LIN {X 0,Y 284.664,Z 673.734,A -85,B 0,C 180,E1 -17037.975,E2 -17037.975} C_VEL
LIN {X 0,Y 285.259,Z 669.776,A -85,B 0,C 180,E1 -17041.157,E2 -17041.157} C_VEL
LIN {X 0,Y 285.946,Z 665.881,A -85,B 0,C 180,E1 -17044.423,E2 -17044.423} C_VEL
LIN {X 0,Y 286.19,Z 663.974,A -85,B 0,C 180,E1 -17046.113,E2 -17046.113} C_VEL
LIN {X 0,Y 286.242,Z 661.735,A -85,B 0,C 180,E1 -17048.216,E2 -17048.216} C_VEL
LIN {X 0,Y 285.887,Z 658.472,A -85,B 0,C 180,E1 -17051.587,E2 -17051.587} C_VEL
LIN {X 0,Y 285.336,Z 655.024,A -85,B 0,C 180,E1 -17055.585,E2 -17055.585} C_VEL
LIN {X 0,Y 284.965,Z 653.006,A -85,B 0,C 180,E1 -17058.249,E2 -17058.249} C_VEL
LIN {X 0,Y 284.54,Z 650.367,A -85,B 0,C 180,E1 -17062.222,E2 -17062.222} C_VEL
LIN {X 0,Y 284.343,Z 649.066,A -85,B 0,C 180,E1 -17064.652,E2 -17064.652} C_VEL
LIN {X 0,Y 284.295,Z 649.074,A -85,B 0,C 180,E1 -17068.726,E2 -17068.726} C_VEL
LIN {X 0,Y 284.396,Z 649.061,A -85,B 0,C 180,E1 -17072.828,E2 -17072.828} C_VEL
LIN {X 0,Y 284.368,Z 649.062,A -85,B 0,C 180,E1 -17076.707,E2 -17076.707} C_VEL
LIN {X 0,Y 284.406,Z 649.059,A -85,B 0,C 180,E1 -17081.262,E2 -17081.262} C_VEL
LIN {X 0,Y 284.494,Z 649.049,A -85,B 0,C 180,E1 -17084.459,E2 -17084.459} C_VEL
LIN {X 0,Y 284.491,Z 649.049,A -85,B 0,C 180,E1 -17088.602,E2 -17088.602} C_VEL
LIN {X 0,Y 284.661,Z 649.027,A -85,B 0,C 180,E1 -17091.481,E2 -17091.481} C_VEL
LIN {X 0,Y 284.604,Z 649.032,A -85,B 0,C 180,E1 -17094.331,E2 -17094.331} C_VEL
LIN {X 0,Y 284.858,Z 649.081,A -85,B 0,C 180,E1 -17098.586,E2 -17098.586} C_VEL
LIN {X 0,Y 285.092,Z 650.526,A -85,B 0,C 180,E1 -17101.413,E2 -17101.413} C_VEL
LIN {X 0,Y 285.18,Z 653.062,A -85,B 0,C 180,E1 -17105.657,E2 -17105.657} C_VEL
LIN {X 0,Y 285.314,Z 654.934,A -85,B 0,C 180,E1 -17108.499,E2 -17108.499} C_VEL
LIN {X 0,Y 284.959,Z 657.078,A -85,B 0,C 180,E1 -17111.38,E2 -17111.38} C_VEL
LIN {X 0,Y 284.349,Z 660.574,A -85,B 0,C 180,E1 -17115.776,E2 -17115.776} C_VEL
LIN {X 0,Y 284.199,Z 661.864,A -85,B 0,C 180,E1 -17117.124,E2 -17117.124} C_VEL
LIN {X 0,Y 285.245,Z 664.861,A -85,B 0,C 180,E1 -17117.428,E2 -17117.428} C_VEL
LIN {X 0,Y 288.856,Z 674.081,A -85,B 0,C 180,E1 -17118.485,E2 -17118.485} C_VEL
LIN {X 0,Y 292.289,Z 685.508,A -85,B 0,C 180,E1 -17119.855,E2 -17119.855} C_VEL
LIN {X 0,Y 294.405,Z 695.768,A -85,B 0,C 180,E1 -17121.173,E2 -17121.173} C_VEL
LIN {X 0,Y 295.274,Z 703.306,A -85,B 0,C 180,E1 -17122.192,E2 -17122.192} C_VEL
LIN {X 0,Y 293.386,Z 714.511,A -85,B 0,C 180,E1 -17123.656,E2 -17123.656} C_VEL
LIN {X 0,Y 291.318,Z 724.902,A -85,B 0,C 180,E1 -17125.354,E2 -17125.354} C_VEL
LIN {X 0,Y 289.305,Z 733.961,A -85,B 0,C 180,E1 -17127.193,E2 -17127.193} C_VEL
LIN {X 0,Y 287.446,Z 742.096,A -85,B 0,C 180,E1 -17129.275,E2 -17129.275} C_VEL
LIN {X 0,Y 285.831,Z 749.014,A -85,B 0,C 180,E1 -17131.5,E2 -17131.5} C_VEL
LIN {X 0,Y 284.513,Z 754.577,A -85,B 0,C 180,E1 -17133.778,E2 -17133.778} C_VEL
LIN {X 0,Y 283.654,Z 758.382,A -85,B 0,C 180,E1 -17135.814,E2 -17135.814} C_VEL
LIN {X 0,Y 282.915,Z 761.858,A -85,B 0,C 180,E1 -17138.392,E2 -17138.392} C_VEL
LIN {X 0,Y 282.479,Z 763.537,A -85,B 0,C 180,E1 -17140.306,E2 -17140.306} C_VEL
LIN {X 0,Y 282.248,Z 764.48,A -85,B 0,C 180,E1 -17142.245,E2 -17142.245} C_VEL
LIN {X 0,Y 282.092,Z 764.707,A -85,B 0,C 180,E1 -17144.234,E2 -17144.234} C_VEL
LIN {X 0,Y 282.099,Z 764.15,A -85,B 0,C 180,E1 -17146.26,E2 -17146.26} C_VEL
LIN {X 0,Y 282.277,Z 762.717,A -85,B 0,C 180,E1 -17148.325,E2 -17148.325} C_VEL
LIN {X 0,Y 282.558,Z 760.336,A -85,B 0,C 180,E1 -17150.449,E2 -17150.449} C_VEL
LIN {X 0,Y 282.955,Z 756.862,A -85,B 0,C 180,E1 -17152.638,E2 -17152.638} C_VEL
LIN {X 0,Y 283.587,Z 752.143,A -85,B 0,C 180,E1 -17154.868,E2 -17154.868} C_VEL
LIN {X 0,Y 284.477,Z 745.924,A -85,B 0,C 180,E1 -17157.137,E2 -17157.137} C_VEL
LIN {X 0,Y 285.721,Z 737.947,A -85,B 0,C 180,E1 -17159.419,E2 -17159.419} C_VEL
LIN {X 0,Y 286.896,Z 730.138,A -85,B 0,C 180,E1 -17161.224,E2 -17161.224} C_VEL
LIN {X 0,Y 288.359,Z 720.685,A -85,B 0,C 180,E1 -17163.004,E2 -17163.004} C_VEL
LIN {X 0,Y 289.993,Z 709.239,A -85,B 0,C 180,E1 -17164.713,E2 -17164.713} C_VEL
LIN {X 0,Y 291.243,Z 698.743,A -85,B 0,C 180,E1 -17165.97,E2 -17165.97} C_VEL
LIN {X 0,Y 289.669,Z 688.156,A -85,B 0,C 180,E1 -17167.157,E2 -17167.157} C_VEL
LIN {X 0,Y 287.141,Z 675.561,A -85,B 0,C 180,E1 -17168.319,E2 -17168.319} C_VEL
LIN {X 0,Y 283.658,Z 661.926,A -85,B 0,C 180,E1 -17169.325,E2 -17169.325} C_VEL
LIN {X 0,Y 283.257,Z 660.019,A -85,B 0,C 180,E1 -17169.437,E2 -17169.437} C_VEL
LIN {X 0,Y 283.549,Z 656.758,A -85,B 0,C 180,E1 -17172.696,E2 -17172.696} C_VEL
LIN {X 0,Y 283.905,Z 653.867,A -85,B 0,C 180,E1 -17175.667,E2 -17175.667} C_VEL
LIN {X 0,Y 284.361,Z 649.706,A -85,B 0,C 180,E1 -17180.037,E2 -17180.037} C_VEL
LIN {X 0,Y 284.468,Z 649.053,A -85,B 0,C 180,E1 -17180.81,E2 -17180.81} C_VEL
LIN {X 0,Y 284.669,Z 649.026,A -85,B 0,C 180,E1 -17182.909,E2 -17182.909} C_VEL
LIN {X 0,Y 284.859,Z 649.001,A -85,B 0,C 180,E1 -17188.586,E2 -17188.586} C_VEL
LIN {X 0,Y 284.859,Z 648.998,A -85,B 0,C 180,E1 -17191.413,E2 -17191.413} C_VEL
LIN {X 0,Y 284.575,Z 649.035,A -85,B 0,C 180,E1 -17195.669,E2 -17195.669} C_VEL
LIN {X 0,Y 284.438,Z 649.054,A -85,B 0,C 180,E1 -17198.758,E2 -17198.758} C_VEL
LIN {X 0,Y 283.86,Z 649.144,A -85,B 0,C 180,E1 -17202.148,E2 -17202.148} C_VEL
LIN {X 0,Y 283.426,Z 653.771,A -85,B 0,C 180,E1 -17205.828,E2 -17205.828} C_VEL
LIN {X 0,Y 283.169,Z 658.716,A -85,B 0,C 180,E1 -17209.686,E2 -17209.686} C_VEL
LIN {X 0,Y 286.493,Z 672.258,A -85,B 0,C 180,E1 -17210.601,E2 -17210.601} C_VEL
LIN {X 0,Y 288.907,Z 683.729,A -85,B 0,C 180,E1 -17211.587,E2 -17211.587} C_VEL
LIN {X 0,Y 290.897,Z 696.161,A -85,B 0,C 180,E1 -17212.904,E2 -17212.904} C_VEL
LIN {X 0,Y 290.964,Z 700.386,A -85,B 0,C 180,E1 -17213.384,E2 -17213.384} C_VEL
LIN {X 0,Y 289.541,Z 711.369,A -85,B 0,C 180,E1 -17214.752,E2 -17214.752} C_VEL
LIN {X 0,Y 287.993,Z 722.2,A -85,B 0,C 180,E1 -17216.446,E2 -17216.446} C_VEL
LIN {X 0,Y 286.526,Z 731.837,A -85,B 0,C 180,E1 -17218.342,E2 -17218.342} C_VEL
LIN {X 0,Y 285.193,Z 740.281,A -85,B 0,C 180,E1 -17220.401,E2 -17220.401} C_VEL
LIN {X 0,Y 284.106,Z 747.82,A -85,B 0,C 180,E1 -17222.747,E2 -17222.747} C_VEL
LIN {X 0,Y 283.266,Z 753.591,A -85,B 0,C 180,E1 -17225.04,E2 -17225.04} C_VEL
LIN {X 0,Y 282.695,Z 757.923,A -85,B 0,C 180,E1 -17227.293,E2 -17227.293} C_VEL
LIN {X 0,Y 282.283,Z 760.988,A -85,B 0,C 180,E1 -17229.483,E2 -17229.483} C_VEL
LIN {X 0,Y 282.008,Z 763.403,A -85,B 0,C 180,E1 -17232.288,E2 -17232.288} C_VEL
LIN {X 0,Y 282.031,Z 764.176,A -85,B 0,C 180,E1 -17234.245,E2 -17234.245} C_VEL
LIN {X 0,Y 282.115,Z 764.191,A -85,B 0,C 180,E1 -17236.255,E2 -17236.255} C_VEL
LIN {X 0,Y 282.358,Z 763.358,A -85,B 0,C 180,E1 -17238.305,E2 -17238.305} C_VEL
LIN {X 0,Y 282.718,Z 761.642,A -85,B 0,C 180,E1 -17240.408,E2 -17240.408} C_VEL
LIN {X 0,Y 283.379,Z 758.988,A -85,B 0,C 180,E1 -17242.524,E2 -17242.524} C_VEL
LIN {X 0,Y 284.183,Z 755.235,A -85,B 0,C 180,E1 -17244.696,E2 -17244.696} C_VEL
LIN {X 0,Y 285.511,Z 749.4,A -85,B 0,C 180,E1 -17247.211,E2 -17247.211} C_VEL
LIN {X 0,Y 287.087,Z 742.446,A -85,B 0,C 180,E1 -17249.499,E2 -17249.499} C_VEL
LIN {X 0,Y 288.904,Z 734.557,A -85,B 0,C 180,E1 -17251.563,E2 -17251.563} C_VEL
LIN {X 0,Y 290.969,Z 725.043,A -85,B 0,C 180,E1 -17253.531,E2 -17253.531} C_VEL
LIN {X 0,Y 292.926,Z 715.188,A -85,B 0,C 180,E1 -17255.167,E2 -17255.167} C_VEL
LIN {X 0,Y 294.891,Z 703.914,A -85,B 0,C 180,E1 -17256.658,E2 -17256.658} C_VEL
LIN {X 0,Y 294.933,Z 701.005,A -85,B 0,C 180,E1 -17257.033,E2 -17257.033} C_VEL
LIN {X 0,Y 293.39,Z 689.863,A -85,B 0,C 180,E1 -17258.473,E2 -17258.473} C_VEL
LIN {X 0,Y 290.907,Z 679.391,A -85,B 0,C 180,E1 -17259.725,E2 -17259.725} C_VEL
LIN {X 0,Y 286.951,Z 667.38,A -85,B 0,C 180,E1 -17261.054,E2 -17261.054} C_VEL
LIN {X 0,Y 284.148,Z 660.229,A -85,B 0,C 180,E1 -17261.804,E2 -17261.804} C_VEL
LIN {X 0,Y 284.051,Z 659.674,A -85,B 0,C 180,E1 -17261.891,E2 -17261.891} C_VEL
LIN {X 0,Y 284.171,Z 658.068,A -85,B 0,C 180,E1 -17263.229,E2 -17263.229} C_VEL
LIN {X 0,Y 283.618,Z 656.803,A -85,B 0,C 180,E1 -17264.387,E2 -17264.387} C_VEL
LIN {X 0,Y 280.968,Z 655.129,A -85,B 0,C 180,E1 -17266.295,E2 -17266.295} C_VEL
LIN {X 0,Y 278.693,Z 653.829,A -85,B 0,C 180,E1 -17267.848,E2 -17267.848} C_VEL
LIN {X 0,Y 277.735,Z 652.691,A -85,B 0,C 180,E1 -17269.04,E2 -17269.04} C_VEL
LIN {X 0,Y 277.669,Z 652.253,A -85,B 0,C 180,E1 -17269.441,E2 -17269.441} C_VEL
LIN {X 0,Y 277.548,Z 649.917,A -85,B 0,C 180,E1 -17271.628,E2 -17271.628} C_VEL
LIN {X 0,Y 277.563,Z 649.914,A -85,B 0,C 180,E1 -17274.187,E2 -17274.187} C_VEL
LIN {X 0,Y 277.82,Z 649.879,A -85,B 0,C 180,E1 -17278.55,E2 -17278.55} C_VEL
LIN {X 0,Y 277.82,Z 649.88,A -85,B 0,C 180,E1 -17281.45,E2 -17281.45} C_VEL
LIN {X 0,Y 277.65,Z 649.899,A -85,B 0,C 180,E1 -17287.271,E2 -17287.271} C_VEL
LIN {X 0,Y 277.503,Z 649.918,A -85,B 0,C 180,E1 -17290.211,E2 -17290.211} C_VEL
LIN {X 0,Y 277.431,Z 649.926,A -85,B 0,C 180,E1 -17294.674,E2 -17294.674} C_VEL
LIN {X 0,Y 277.341,Z 649.936,A -85,B 0,C 180,E1 -17299.234,E2 -17299.234} C_VEL
LIN {X 0,Y 277.316,Z 649.94,A -85,B 0,C 180,E1 -17304.171,E2 -17304.171} C_VEL
LIN {X 0,Y 277.323,Z 649.942,A -85,B 0,C 180,E1 -17307.506,E2 -17307.506} C_VEL
LIN {X 0,Y 277.269,Z 649.947,A -85,B 0,C 180,E1 -17310.482,E2 -17310.482} C_VEL
LIN {X 0,Y 277.244,Z 649.95,A -85,B 0,C 180,E1 -17313.896,E2 -17313.896} C_VEL
LIN {X 0,Y 277.265,Z 649.946,A -85,B 0,C 180,E1 -17317.47,E2 -17317.47} C_VEL
LIN {X 0,Y 277.207,Z 649.956,A -85,B 0,C 180,E1 -17321.237,E2 -17321.237} C_VEL
LIN {X 0,Y 277.273,Z 650.135,A -85,B 0,C 180,E1 -17324.659,E2 -17324.659} C_VEL
LIN {X 0,Y 278.128,Z 654.82,A -85,B 0,C 180,E1 -17328.93,E2 -17328.93} C_VEL
LIN {X 0,Y 278.627,Z 657.699,A -85,B 0,C 180,E1 -17331.438,E2 -17331.438} C_VEL
LIN {X 0,Y 278.8,Z 660.491,A -85,B 0,C 180,E1 -17333.771,E2 -17333.771} C_VEL
LIN {X 0,Y 278.36,Z 663.849,A -85,B 0,C 180,E1 -17336.427,E2 -17336.427} C_VEL
LIN {X 0,Y 277.598,Z 669.016,A -85,B 0,C 180,E1 -17340.418,E2 -17340.418} C_VEL
LIN {X 0,Y 277.426,Z 670.534,A -85,B 0,C 180,E1 -17341.447,E2 -17341.447} C_VEL
LIN {X 0,Y 278.249,Z 673.76,A -85,B 0,C 180,E1 -17341.713,E2 -17341.713} C_VEL
LIN {X 0,Y 281.779,Z 685.347,A -85,B 0,C 180,E1 -17342.86,E2 -17342.86} C_VEL
LIN {X 0,Y 284.486,Z 697.852,A -85,B 0,C 180,E1 -17344.193,E2 -17344.193} C_VEL
LIN {X 0,Y 285.824,Z 708.755,A -85,B 0,C 180,E1 -17345.475,E2 -17345.475} C_VEL
LIN {X 0,Y 286.188,Z 719.399,A -85,B 0,C 180,E1 -17346.865,E2 -17346.865} C_VEL
LIN {X 0,Y 285.951,Z 725.836,A -85,B 0,C 180,E1 -17347.798,E2 -17347.798} C_VEL
LIN {X 0,Y 283.945,Z 735.872,A -85,B 0,C 180,E1 -17349.348,E2 -17349.348} C_VEL
LIN {X 0,Y 281.936,Z 744.978,A -85,B 0,C 180,E1 -17351.092,E2 -17351.092} C_VEL
LIN {X 0,Y 280.014,Z 753.864,A -85,B 0,C 180,E1 -17353.224,E2 -17353.224} C_VEL
LIN {X 0,Y 278.44,Z 761.082,A -85,B 0,C 180,E1 -17355.381,E2 -17355.381} C_VEL
LIN {X 0,Y 277.093,Z 766.88,A -85,B 0,C 180,E1 -17357.551,E2 -17357.551} C_VEL
LIN {X 0,Y 276.211,Z 771.449,A -85,B 0,C 180,E1 -17359.741,E2 -17359.741} C_VEL
LIN {X 0,Y 275.813,Z 773.863,A -85,B 0,C 180,E1 -17361.206,E2 -17361.206} C_VEL
LIN {X 0,Y 275.509,Z 775.851,A -85,B 0,C 180,E1 -17362.673,E2 -17362.673} C_VEL
LIN {X 0,Y 275.326,Z 777.779,A -85,B 0,C 180,E1 -17364.575,E2 -17364.575} C_VEL
LIN {X 0,Y 275.265,Z 780.485,A -85,B 0,C 180,E1 -17368.538,E2 -17368.538} C_VEL
LIN {X 0,Y 275.28,Z 781.022,A -85,B 0,C 180,E1 -17370.001,E2 -17370.001} C_VEL
LIN {X 0,Y 275.262,Z 781.121,A -85,B 0,C 180,E1 -17371.464,E2 -17371.464} C_VEL
LIN {X 0,Y 275.257,Z 780.809,A -85,B 0,C 180,E1 -17372.928,E2 -17372.928} C_VEL
LIN {X 0,Y 275.379,Z 779.015,A -85,B 0,C 180,E1 -17375.86,E2 -17375.86} C_VEL
LIN {X 0,Y 275.531,Z 777.483,A -85,B 0,C 180,E1 -17377.328,E2 -17377.328} C_VEL
LIN {X 0,Y 276.016,Z 774.394,A -85,B 0,C 180,E1 -17379.527,E2 -17379.527} C_VEL
LIN {X 0,Y 276.843,Z 770.267,A -85,B 0,C 180,E1 -17381.718,E2 -17381.718} C_VEL
LIN {X 0,Y 278.211,Z 763.998,A -85,B 0,C 180,E1 -17384.259,E2 -17384.259} C_VEL
LIN {X 0,Y 279.916,Z 757.219,A -85,B 0,C 180,E1 -17386.408,E2 -17386.408} C_VEL
LIN {X 0,Y 281.667,Z 748.963,A -85,B 0,C 180,E1 -17388.53,E2 -17388.53} C_VEL
LIN {X 0,Y 283.596,Z 740.359,A -85,B 0,C 180,E1 -17390.301,E2 -17390.301} C_VEL
LIN {X 0,Y 285.822,Z 729.966,A -85,B 0,C 180,E1 -17392.023,E2 -17392.023} C_VEL
LIN {X 0,Y 286.844,Z 723.901,A -85,B 0,C 180,E1 -17392.89,E2 -17392.89} C_VEL
LIN {X 0,Y 286.621,Z 713.07,A -85,B 0,C 180,E1 -17394.404,E2 -17394.404} C_VEL
LIN {X 0,Y 285.273,Z 701.307,A -85,B 0,C 180,E1 -17395.863,E2 -17395.863} C_VEL
LIN {X 0,Y 282.516,Z 688.923,A -85,B 0,C 180,E1 -17397.285,E2 -17397.285} C_VEL
LIN {X 0,Y 279.072,Z 677.521,A -85,B 0,C 180,E1 -17398.511,E2 -17398.511} C_VEL
LIN {X 0,Y 277.896,Z 674.354,A -85,B 0,C 180,E1 -17398.849,E2 -17398.849} C_VEL
LIN {X 0,Y 277.781,Z 673.521,A -85,B 0,C 180,E1 -17398.939,E2 -17398.939} C_VEL
LIN {X 0,Y 278.409,Z 669.828,A -85,B 0,C 180,E1 -17402.014,E2 -17402.014} C_VEL
LIN {X 0,Y 279.079,Z 665.982,A -85,B 0,C 180,E1 -17405.395,E2 -17405.395} C_VEL
LIN {X 0,Y 279.227,Z 664.096,A -85,B 0,C 180,E1 -17407.162,E2 -17407.162} C_VEL
LIN {X 0,Y 279.168,Z 662.256,A -85,B 0,C 180,E1 -17409.004,E2 -17409.004} C_VEL
LIN {X 0,Y 279.005,Z 660.453,A -85,B 0,C 180,E1 -17410.915,E2 -17410.915} C_VEL
LIN {X 0,Y 278.478,Z 656.993,A -85,B 0,C 180,E1 -17414.963,E2 -17414.963} C_VEL
LIN {X 0,Y 277.945,Z 654.091,A -85,B 0,C 180,E1 -17418.896,E2 -17418.896} C_VEL
LIN {X 0,Y 277.569,Z 651.765,A -85,B 0,C 180,E1 -17422.578,E2 -17422.578} C_VEL
LIN {X 0,Y 277.249,Z 649.949,A -85,B 0,C 180,E1 -17426.104,E2 -17426.104} C_VEL
LIN {X 0,Y 277.263,Z 649.946,A -85,B 0,C 180,E1 -17429.539,E2 -17429.539} C_VEL
LIN {X 0,Y 277.358,Z 649.938,A -85,B 0,C 180,E1 -17432.864,E2 -17432.864} C_VEL
LIN {X 0,Y 277.33,Z 649.936,A -85,B 0,C 180,E1 -17436.08,E2 -17436.08} C_VEL
LIN {X 0,Y 277.347,Z 649.939,A -85,B 0,C 180,E1 -17440.766,E2 -17440.766} C_VEL
LIN {X 0,Y 277.437,Z 649.928,A -85,B 0,C 180,E1 -17445.326,E2 -17445.326} C_VEL
LIN {X 0,Y 277.509,Z 649.915,A -85,B 0,C 180,E1 -17449.789,E2 -17449.789} C_VEL
LIN {X 0,Y 277.655,Z 649.898,A -85,B 0,C 180,E1 -17452.729,E2 -17452.729} C_VEL
LIN {X 0,Y 277.701,Z 649.921,A -85,B 0,C 180,E1 -17457.099,E2 -17457.099} C_VEL
LIN {X 0,Y 278.1,Z 651.215,A -85,B 0,C 180,E1 -17460,E2 -17460} C_VEL
LIN {X 0,Y 278.154,Z 652.769,A -85,B 0,C 180,E1 -17462.897,E2 -17462.897} C_VEL
LIN {X 0,Y 278.298,Z 655.402,A -85,B 0,C 180,E1 -17467.254,E2 -17467.254} C_VEL
LIN {X 0,Y 278.127,Z 657.42,A -85,B 0,C 180,E1 -17470.188,E2 -17470.188} C_VEL
LIN {X 0,Y 277.464,Z 660.842,A -85,B 0,C 180,E1 -17474.673,E2 -17474.673} C_VEL
LIN {X 0,Y 277.293,Z 661.957,A -85,B 0,C 180,E1 -17476.092,E2 -17476.092} C_VEL
LIN {X 0,Y 278.408,Z 665.25,A -85,B 0,C 180,E1 -17476.461,E2 -17476.461} C_VEL
LIN {X 0,Y 282.09,Z 674.295,A -85,B 0,C 180,E1 -17477.583,E2 -17477.583} C_VEL
LIN {X 0,Y 285.242,Z 684.375,A -85,B 0,C 180,E1 -17478.858,E2 -17478.858} C_VEL
LIN {X 0,Y 287.762,Z 695.631,A -85,B 0,C 180,E1 -17480.367,E2 -17480.367} C_VEL
LIN {X 0,Y 288.826,Z 704.29,A -85,B 0,C 180,E1 -17481.603,E2 -17481.603} C_VEL
LIN {X 0,Y 286.967,Z 715.061,A -85,B 0,C 180,E1 -17483.07,E2 -17483.07} C_VEL
LIN {X 0,Y 284.798,Z 725.402,A -85,B 0,C 180,E1 -17484.804,E2 -17484.804} C_VEL
LIN {X 0,Y 282.782,Z 733.953,A -85,B 0,C 180,E1 -17486.574,E2 -17486.574} C_VEL
LIN {X 0,Y 280.712,Z 742.491,A -85,B 0,C 180,E1 -17488.803,E2 -17488.803} C_VEL
LIN {X 0,Y 279.007,Z 749.379,A -85,B 0,C 180,E1 -17491.081,E2 -17491.081} C_VEL
LIN {X 0,Y 277.637,Z 754.755,A -85,B 0,C 180,E1 -17493.347,E2 -17493.347} C_VEL
LIN {X 0,Y 276.601,Z 759.08,A -85,B 0,C 180,E1 -17495.76,E2 -17495.76} C_VEL
LIN {X 0,Y 275.965,Z 761.825,A -85,B 0,C 180,E1 -17497.863,E2 -17497.863} C_VEL
LIN {X 0,Y 275.429,Z 763.743,A -85,B 0,C 180,E1 -17500.048,E2 -17500.048} C_VEL
LIN {X 0,Y 275.156,Z 764.744,A -85,B 0,C 180,E1 -17502.207,E2 -17502.207} C_VEL
LIN {X 0,Y 274.99,Z 764.896,A -85,B 0,C 180,E1 -17504.307,E2 -17504.307} C_VEL
LIN {X 0,Y 275.004,Z 764.257,A -85,B 0,C 180,E1 -17506.368,E2 -17506.368} C_VEL
LIN {X 0,Y 275.184,Z 762.849,A -85,B 0,C 180,E1 -17508.392,E2 -17508.392} C_VEL
LIN {X 0,Y 275.465,Z 760.673,A -85,B 0,C 180,E1 -17510.369,E2 -17510.369} C_VEL
LIN {X 0,Y 275.781,Z 757.799,A -85,B 0,C 180,E1 -17512.293,E2 -17512.293} C_VEL
LIN {X 0,Y 276.374,Z 753.558,A -85,B 0,C 180,E1 -17514.463,E2 -17514.463} C_VEL
LIN {X 0,Y 277.188,Z 747.684,A -85,B 0,C 180,E1 -17516.794,E2 -17516.794} C_VEL
LIN {X 0,Y 278.419,Z 740.212,A -85,B 0,C 180,E1 -17519.121,E2 -17519.121} C_VEL
LIN {X 0,Y 279.643,Z 732.382,A -85,B 0,C 180,E1 -17521.067,E2 -17521.067} C_VEL
LIN {X 0,Y 281.228,Z 722.404,A -85,B 0,C 180,E1 -17523.066,E2 -17523.066} C_VEL
LIN {X 0,Y 282.664,Z 712.862,A -85,B 0,C 180,E1 -17524.611,E2 -17524.611} C_VEL
LIN {X 0,Y 284.064,Z 702.39,A -85,B 0,C 180,E1 -17525.984,E2 -17525.984} C_VEL
LIN {X 0,Y 284.159,Z 697.909,A -85,B 0,C 180,E1 -17526.515,E2 -17526.515} C_VEL
LIN {X 0,Y 282.167,Z 685.765,A -85,B 0,C 180,E1 -17527.869,E2 -17527.869} C_VEL
LIN {X 0,Y 279.45,Z 672.872,A -85,B 0,C 180,E1 -17529.047,E2 -17529.047} C_VEL
LIN {X 0,Y 276.243,Z 660.167,A -85,B 0,C 180,E1 -17529.994,E2 -17529.994} C_VEL
LIN {X 0,Y 276.595,Z 656.508,A -85,B 0,C 180,E1 -17533.769,E2 -17533.769} C_VEL
LIN {X 0,Y 276.918,Z 653.626,A -85,B 0,C 180,E1 -17536.796,E2 -17536.796} C_VEL
LIN {X 0,Y 277.495,Z 649.921,A -85,B 0,C 180,E1 -17541.02,E2 -17541.02} C_VEL
LIN {X 0,Y 277.565,Z 649.908,A -85,B 0,C 180,E1 -17544.186,E2 -17544.186} C_VEL
LIN {X 0,Y 277.825,Z 649.876,A -85,B 0,C 180,E1 -17548.55,E2 -17548.55} C_VEL
LIN {X 0,Y 277.824,Z 649.874,A -85,B 0,C 180,E1 -17551.449,E2 -17551.449} C_VEL
LIN {X 0,Y 277.54,Z 649.912,A -85,B 0,C 180,E1 -17555.813,E2 -17555.813} C_VEL
LIN {X 0,Y 277.372,Z 649.934,A -85,B 0,C 180,E1 -17558.818,E2 -17558.818} C_VEL
LIN {X 0,Y 276.837,Z 650.016,A -85,B 0,C 180,E1 -17562.089,E2 -17562.089} C_VEL
LIN {X 0,Y 276.314,Z 655.191,A -85,B 0,C 180,E1 -17566.247,E2 -17566.247} C_VEL
LIN {X 0,Y 276.146,Z 658.767,A -85,B 0,C 180,E1 -17569.127,E2 -17569.127} C_VEL
LIN {X 0,Y 279.856,Z 674,A -85,B 0,C 180,E1 -17570.235,E2 -17570.235} C_VEL
LIN {X 0,Y 282.29,Z 686.105,A -85,B 0,C 180,E1 -17571.352,E2 -17571.352} C_VEL
LIN {X 0,Y 284.209,Z 698.375,A -85,B 0,C 180,E1 -17572.729,E2 -17572.729} C_VEL
LIN {X 0,Y 283.1,Z 708.767,A -85,B 0,C 180,E1 -17573.995,E2 -17573.995} C_VEL
LIN {X 0,Y 281.417,Z 720.109,A -85,B 0,C 180,E1 -17575.723,E2 -17575.723} C_VEL
LIN {X 0,Y 280.011,Z 729.296,A -85,B 0,C 180,E1 -17577.463,E2 -17577.463} C_VEL
LIN {X 0,Y 278.625,Z 737.842,A -85,B 0,C 180,E1 -17579.462,E2 -17579.462} C_VEL
LIN {X 0,Y 277.423,Z 745.682,A -85,B 0,C 180,E1 -17581.768,E2 -17581.768} C_VEL
LIN {X 0,Y 276.548,Z 751.68,A -85,B 0,C 180,E1 -17583.992,E2 -17583.992} C_VEL
LIN {X 0,Y 275.946,Z 755.669,A -85,B 0,C 180,E1 -17585.857,E2 -17585.857} C_VEL
LIN {X 0,Y 275.32,Z 760.235,A -85,B 0,C 180,E1 -17588.711,E2 -17588.711} C_VEL
LIN {X 0,Y 274.944,Z 763.169,A -85,B 0,C 180,E1 -17591.651,E2 -17591.651} C_VEL
LIN {X 0,Y 274.933,Z 764.369,A -85,B 0,C 180,E1 -17594.295,E2 -17594.295} C_VEL
LIN {X 0,Y 275.026,Z 764.404,A -85,B 0,C 180,E1 -17596.373,E2 -17596.373} C_VEL
LIN {X 0,Y 275.275,Z 763.625,A -85,B 0,C 180,E1 -17598.409,E2 -17598.409} C_VEL
LIN {X 0,Y 275.622,Z 762.123,A -85,B 0,C 180,E1 -17600.396,E2 -17600.396} C_VEL
LIN {X 0,Y 276.256,Z 759.873,A -85,B 0,C 180,E1 -17602.369,E2 -17602.369} C_VEL
LIN {X 0,Y 276.943,Z 756.914,A -85,B 0,C 180,E1 -17604.297,E2 -17604.297} C_VEL
LIN {X 0,Y 278.024,Z 752.404,A -85,B 0,C 180,E1 -17606.53,E2 -17606.53} C_VEL
LIN {X 0,Y 279.445,Z 746.551,A -85,B 0,C 180,E1 -17608.769,E2 -17608.769} C_VEL
LIN {X 0,Y 281.274,Z 739.196,A -85,B 0,C 180,E1 -17610.987,E2 -17610.987} C_VEL
LIN {X 0,Y 283.167,Z 731.129,A -85,B 0,C 180,E1 -17612.942,E2 -17612.942} C_VEL
LIN {X 0,Y 285.089,Z 722.466,A -85,B 0,C 180,E1 -17614.638,E2 -17614.638} C_VEL
LIN {X 0,Y 287.35,Z 711.258,A -85,B 0,C 180,E1 -17616.39,E2 -17616.39} C_VEL
LIN {X 0,Y 288.529,Z 704.525,A -85,B 0,C 180,E1 -17617.27,E2 -17617.27} C_VEL
LIN {X 0,Y 287.71,Z 695.7,A -85,B 0,C 180,E1 -17618.505,E2 -17618.505} C_VEL
LIN {X 0,Y 285.726,Z 685.274,A -85,B 0,C 180,E1 -17619.857,E2 -17619.857} C_VEL
LIN {X 0,Y 282.201,Z 673.271,A -85,B 0,C 180,E1 -17621.315,E2 -17621.315} C_VEL
LIN {X 0,Y 278.28,Z 663.164,A -85,B 0,C 180,E1 -17622.501,E2 -17622.501} C_VEL
LIN {X 0,Y 277.194,Z 659.893,A -85,B 0,C 180,E1 -17622.858,E2 -17622.858} C_VEL
LIN {X 0,Y 277.622,Z 655.249,A -85,B 0,C 180,E1 -17626.83,E2 -17626.83} C_VEL
LIN {X 0,Y 277.669,Z 652.253,A -85,B 0,C 180,E1 -17629.441,E2 -17629.441} C_VEL
LIN {X 0,Y 276.986,Z 651.242,A -85,B 0,C 180,E1 -17630.631,E2 -17630.631} C_VEL
LIN {X 0,Y 275.333,Z 650.76,A -85,B 0,C 180,E1 -17631.812,E2 -17631.812} C_VEL
LIN {X 0,Y 271.5,Z 650.708,A -85,B 0,C 180,E1 -17634.203,E2 -17634.203} C_VEL
LIN {X 0,Y 270.496,Z 650.794,A -85,B 0,C 180,E1 -17635.453,E2 -17635.453} C_VEL
LIN {X 0,Y 270.452,Z 650.797,A -85,B 0,C 180,E1 -17635.876,E2 -17635.876} C_VEL
LIN {X 0,Y 270.785,Z 650.756,A -85,B 0,C 180,E1 -17638.513,E2 -17638.513} C_VEL
LIN {X 0,Y 270.785,Z 650.756,A -85,B 0,C 180,E1 -17641.487,E2 -17641.487} C_VEL
LIN {X 0,Y 270.608,Z 650.776,A -85,B 0,C 180,E1 -17647.461,E2 -17647.461} C_VEL
LIN {X 0,Y 270.438,Z 650.799,A -85,B 0,C 180,E1 -17650.481,E2 -17650.481} C_VEL
LIN {X 0,Y 270.4,Z 650.804,A -85,B 0,C 180,E1 -17655.065,E2 -17655.065} C_VEL
LIN {X 0,Y 270.298,Z 650.816,A -85,B 0,C 180,E1 -17659.756,E2 -17659.756} C_VEL
LIN {X 0,Y 270.271,Z 650.819,A -85,B 0,C 180,E1 -17664.586,E2 -17664.586} C_VEL
LIN {X 0,Y 270.267,Z 650.819,A -85,B 0,C 180,E1 -17667.909,E2 -17667.909} C_VEL
LIN {X 0,Y 270.181,Z 650.829,A -85,B 0,C 180,E1 -17671.349,E2 -17671.349} C_VEL
LIN {X 0,Y 270.199,Z 650.828,A -85,B 0,C 180,E1 -17674.906,E2 -17674.906} C_VEL
LIN {X 0,Y 270.195,Z 650.83,A -85,B 0,C 180,E1 -17678.711,E2 -17678.711} C_VEL
LIN {X 0,Y 270.169,Z 650.833,A -85,B 0,C 180,E1 -17683.251,E2 -17683.251} C_VEL
LIN {X 0,Y 270.201,Z 650.842,A -85,B 0,C 180,E1 -17684.235,E2 -17684.235} C_VEL
LIN {X 0,Y 270.815,Z 654.374,A -85,B 0,C 180,E1 -17687.568,E2 -17687.568} C_VEL
LIN {X 0,Y 271.542,Z 658.087,A -85,B 0,C 180,E1 -17690.937,E2 -17690.937} C_VEL
LIN {X 0,Y 271.755,Z 661.07,A -85,B 0,C 180,E1 -17693.502,E2 -17693.502} C_VEL
LIN {X 0,Y 271.398,Z 664.087,A -85,B 0,C 180,E1 -17695.961,E2 -17695.961} C_VEL
LIN {X 0,Y 270.547,Z 669.692,A -85,B 0,C 180,E1 -17700.366,E2 -17700.366} C_VEL
LIN {X 0,Y 271.416,Z 673.063,A -85,B 0,C 180,E1 -17700.657,E2 -17700.657} C_VEL
LIN {X 0,Y 274.431,Z 682.408,A -85,B 0,C 180,E1 -17701.635,E2 -17701.635} C_VEL
LIN {X 0,Y 277.348,Z 694.66,A -85,B 0,C 180,E1 -17703,E2 -17703} C_VEL
LIN {X 0,Y 279.191,Z 706.952,A -85,B 0,C 180,E1 -17704.484,E2 -17704.484} C_VEL
LIN {X 0,Y 279.671,Z 717.565,A -85,B 0,C 180,E1 -17705.895,E2 -17705.895} C_VEL
LIN {X 0,Y 279.433,Z 726.583,A -85,B 0,C 180,E1 -17707.252,E2 -17707.252} C_VEL
LIN {X 0,Y 277.349,Z 736.427,A -85,B 0,C 180,E1 -17708.833,E2 -17708.833} C_VEL
LIN {X 0,Y 275.258,Z 745.382,A -85,B 0,C 180,E1 -17710.615,E2 -17710.615} C_VEL
LIN {X 0,Y 273.517,Z 752.815,A -85,B 0,C 180,E1 -17712.428,E2 -17712.428} C_VEL
LIN {X 0,Y 271.831,Z 760.152,A -85,B 0,C 180,E1 -17714.633,E2 -17714.633} C_VEL
LIN {X 0,Y 270.145,Z 766.95,A -85,B 0,C 180,E1 -17717.225,E2 -17717.225} C_VEL
LIN {X 0,Y 269.212,Z 771.455,A -85,B 0,C 180,E1 -17719.471,E2 -17719.471} C_VEL
LIN {X 0,Y 268.762,Z 773.84,A -85,B 0,C 180,E1 -17720.974,E2 -17720.974} C_VEL
LIN {X 0,Y 268.448,Z 775.8,A -85,B 0,C 180,E1 -17722.479,E2 -17722.479} C_VEL
LIN {X 0,Y 268.224,Z 777.859,A -85,B 0,C 180,E1 -17724.671,E2 -17724.671} C_VEL
LIN {X 0,Y 268.191,Z 780.206,A -85,B 0,C 180,E1 -17728.499,E2 -17728.499} C_VEL
LIN {X 0,Y 268.203,Z 780.769,A -85,B 0,C 180,E1 -17730.001,E2 -17730.001} C_VEL
LIN {X 0,Y 268.188,Z 780.919,A -85,B 0,C 180,E1 -17731.502,E2 -17731.502} C_VEL
LIN {X 0,Y 268.17,Z 780.632,A -85,B 0,C 180,E1 -17733.005,E2 -17733.005} C_VEL
LIN {X 0,Y 268.301,Z 778.889,A -85,B 0,C 180,E1 -17736.015,E2 -17736.015} C_VEL
LIN {X 0,Y 268.484,Z 777.415,A -85,B 0,C 180,E1 -17737.521,E2 -17737.521} C_VEL
LIN {X 0,Y 268.992,Z 774.385,A -85,B 0,C 180,E1 -17739.778,E2 -17739.778} C_VEL
LIN {X 0,Y 269.865,Z 770.328,A -85,B 0,C 180,E1 -17742.026,E2 -17742.026} C_VEL
LIN {X 0,Y 271.341,Z 764.143,A -85,B 0,C 180,E1 -17744.628,E2 -17744.628} C_VEL
LIN {X 0,Y 273.116,Z 757.441,A -85,B 0,C 180,E1 -17746.828,E2 -17746.828} C_VEL
LIN {X 0,Y 275.104,Z 748.701,A -85,B 0,C 180,E1 -17749.139,E2 -17749.139} C_VEL
LIN {X 0,Y 276.987,Z 740.86,A -85,B 0,C 180,E1 -17750.808,E2 -17750.808} C_VEL
LIN {X 0,Y 279.302,Z 730.676,A -85,B 0,C 180,E1 -17752.566,E2 -17752.566} C_VEL
LIN {X 0,Y 280.322,Z 724.734,A -85,B 0,C 180,E1 -17753.454,E2 -17753.454} C_VEL
LIN {X 0,Y 280.168,Z 714.231,A -85,B 0,C 180,E1 -17754.994,E2 -17754.994} C_VEL
LIN {X 0,Y 278.898,Z 702.195,A -85,B 0,C 180,E1 -17756.573,E2 -17756.573} C_VEL
LIN {X 0,Y 276.314,Z 690.335,A -85,B 0,C 180,E1 -17758.033,E2 -17758.033} C_VEL
LIN {X 0,Y 273.401,Z 680.637,A -85,B 0,C 180,E1 -17759.169,E2 -17759.169} C_VEL
LIN {X 0,Y 271.104,Z 674.101,A -85,B 0,C 180,E1 -17759.903,E2 -17759.903} C_VEL
LIN {X 0,Y 270.983,Z 673.243,A -85,B 0,C 180,E1 -17760.004,E2 -17760.004} C_VEL
LIN {X 0,Y 271.869,Z 668.492,A -85,B 0,C 180,E1 -17764.185,E2 -17764.185} C_VEL
LIN {X 0,Y 272.229,Z 665.678,A -85,B 0,C 180,E1 -17766.84,E2 -17766.84} C_VEL
LIN {X 0,Y 272.076,Z 662.437,A -85,B 0,C 180,E1 -17770.224,E2 -17770.224} C_VEL
LIN {X 0,Y 271.586,Z 658.961,A -85,B 0,C 180,E1 -17774.323,E2 -17774.323} C_VEL
LIN {X 0,Y 271.046,Z 655.722,A -85,B 0,C 180,E1 -17778.76,E2 -17778.76} C_VEL
LIN {X 0,Y 270.775,Z 654.007,A -85,B 0,C 180,E1 -17781.47,E2 -17781.47} C_VEL
LIN {X 0,Y 270.432,Z 652.044,A -85,B 0,C 180,E1 -17785.128,E2 -17785.128} C_VEL
LIN {X 0,Y 270.28,Z 651.233,A -85,B 0,C 180,E1 -17786.903,E2 -17786.903} C_VEL
LIN {X 0,Y 270.202,Z 650.827,A -85,B 0,C 180,E1 -17789.131,E2 -17789.131} C_VEL
LIN {X 0,Y 270.265,Z 650.818,A -85,B 0,C 180,E1 -17792.146,E2 -17792.146} C_VEL
LIN {X 0,Y 270.279,Z 650.816,A -85,B 0,C 180,E1 -17795.519,E2 -17795.519} C_VEL
LIN {X 0,Y 270.304,Z 650.815,A -85,B 0,C 180,E1 -17800.245,E2 -17800.245} C_VEL
LIN {X 0,Y 270.405,Z 650.803,A -85,B 0,C 180,E1 -17804.936,E2 -17804.936} C_VEL
LIN {X 0,Y 270.444,Z 650.796,A -85,B 0,C 180,E1 -17809.519,E2 -17809.519} C_VEL
LIN {X 0,Y 270.613,Z 650.775,A -85,B 0,C 180,E1 -17812.539,E2 -17812.539} C_VEL
LIN {X 0,Y 270.433,Z 650.87,A -85,B 0,C 180,E1 -17815.528,E2 -17815.528} C_VEL
LIN {X 0,Y 270.979,Z 652.01,A -85,B 0,C 180,E1 -17818.514,E2 -17818.514} C_VEL
LIN {X 0,Y 271.181,Z 653.418,A -85,B 0,C 180,E1 -17821.485,E2 -17821.485} C_VEL
LIN {X 0,Y 271.271,Z 655.921,A -85,B 0,C 180,E1 -17825.948,E2 -17825.948} C_VEL
LIN {X 0,Y 271.304,Z 657.812,A -85,B 0,C 180,E1 -17828.942,E2 -17828.942} C_VEL
LIN {X 0,Y 270.843,Z 659.975,A -85,B 0,C 180,E1 -17831.981,E2 -17831.981} C_VEL
LIN {X 0,Y 270.409,Z 662.261,A -85,B 0,C 180,E1 -17835.016,E2 -17835.016} C_VEL
LIN {X 0,Y 271.588,Z 665.554,A -85,B 0,C 180,E1 -17835.414,E2 -17835.414} C_VEL
LIN {X 0,Y 276.27,Z 677.077,A -85,B 0,C 180,E1 -17836.961,E2 -17836.961} C_VEL
LIN {X 0,Y 279.278,Z 687.212,A -85,B 0,C 180,E1 -17838.334,E2 -17838.334} C_VEL
LIN {X 0,Y 281.47,Z 697.584,A -85,B 0,C 180,E1 -17839.82,E2 -17839.82} C_VEL
LIN {X 0,Y 282.395,Z 706.444,A -85,B 0,C 180,E1 -17841.153,E2 -17841.153} C_VEL
LIN {X 0,Y 280.212,Z 717.357,A -85,B 0,C 180,E1 -17842.706,E2 -17842.706} C_VEL
LIN {X 0,Y 277.99,Z 727.251,A -85,B 0,C 180,E1 -17844.476,E2 -17844.476} C_VEL
LIN {X 0,Y 275.746,Z 736.128,A -85,B 0,C 180,E1 -17846.455,E2 -17846.455} C_VEL
LIN {X 0,Y 273.714,Z 744.019,A -85,B 0,C 180,E1 -17848.653,E2 -17848.653} C_VEL
LIN {X 0,Y 271.866,Z 750.992,A -85,B 0,C 180,E1 -17851.133,E2 -17851.133} C_VEL
LIN {X 0,Y 270.36,Z 756.515,A -85,B 0,C 180,E1 -17853.711,E2 -17853.711} C_VEL
LIN {X 0,Y 269.419,Z 760.212,A -85,B 0,C 180,E1 -17856.034,E2 -17856.034} C_VEL
LIN {X 0,Y 268.602,Z 763.324,A -85,B 0,C 180,E1 -17858.9,E2 -17858.9} C_VEL
LIN {X 0,Y 268.199,Z 764.587,A -85,B 0,C 180,E1 -17860.928,E2 -17860.928} C_VEL
LIN {X 0,Y 267.98,Z 765.131,A -85,B 0,C 180,E1 -17862.99,E2 -17862.99} C_VEL
LIN {X 0,Y 267.877,Z 764.933,A -85,B 0,C 180,E1 -17865.103,E2 -17865.103} C_VEL
LIN {X 0,Y 267.984,Z 763.921,A -85,B 0,C 180,E1 -17867.249,E2 -17867.249} C_VEL
LIN {X 0,Y 268.349,Z 761.025,A -85,B 0,C 180,E1 -17870.272,E2 -17870.272} C_VEL
LIN {X 0,Y 268.861,Z 756.854,A -85,B 0,C 180,E1 -17873.042,E2 -17873.042} C_VEL
LIN {X 0,Y 269.681,Z 751.075,A -85,B 0,C 180,E1 -17875.756,E2 -17875.756} C_VEL
LIN {X 0,Y 270.844,Z 743.977,A -85,B 0,C 180,E1 -17878.3,E2 -17878.3} C_VEL
LIN {X 0,Y 272.203,Z 735.644,A -85,B 0,C 180,E1 -17880.622,E2 -17880.622} C_VEL
LIN {X 0,Y 273.525,Z 727.533,A -85,B 0,C 180,E1 -17882.451,E2 -17882.451} C_VEL
LIN {X 0,Y 275.118,Z 717.691,A -85,B 0,C 180,E1 -17884.261,E2 -17884.261} C_VEL
LIN {X 0,Y 276.658,Z 707.139,A -85,B 0,C 180,E1 -17885.818,E2 -17885.818} C_VEL
LIN {X 0,Y 277.398,Z 699.786,A -85,B 0,C 180,E1 -17886.729,E2 -17886.729} C_VEL
LIN {X 0,Y 275.62,Z 688.276,A -85,B 0,C 180,E1 -17888.104,E2 -17888.104} C_VEL
LIN {X 0,Y 272.966,Z 675.258,A -85,B 0,C 180,E1 -17889.373,E2 -17889.373} C_VEL
LIN {X 0,Y 269.623,Z 662.25,A -85,B 0,C 180,E1 -17890.39,E2 -17890.39} C_VEL
LIN {X 0,Y 269.254,Z 660.353,A -85,B 0,C 180,E1 -17890.561,E2 -17890.561} C_VEL
LIN {X 0,Y 269.691,Z 656.242,A -85,B 0,C 180,E1 -17894.894,E2 -17894.894} C_VEL
LIN {X 0,Y 270.187,Z 652.025,A -85,B 0,C 180,E1 -17899.508,E2 -17899.508} C_VEL
LIN {X 0,Y 270.442,Z 650.799,A -85,B 0,C 180,E1 -17901.029,E2 -17901.029} C_VEL
LIN {X 0,Y 270.534,Z 650.784,A -85,B 0,C 180,E1 -17904.035,E2 -17904.035} C_VEL
LIN {X 0,Y 270.79,Z 650.752,A -85,B 0,C 180,E1 -17908.512,E2 -17908.512} C_VEL
LIN {X 0,Y 270.79,Z 650.75,A -85,B 0,C 180,E1 -17911.487,E2 -17911.487} C_VEL
LIN {X 0,Y 270.506,Z 650.788,A -85,B 0,C 180,E1 -17915.965,E2 -17915.965} C_VEL
LIN {X 0,Y 270.301,Z 650.816,A -85,B 0,C 180,E1 -17918.974,E2 -17918.974} C_VEL
LIN {X 0,Y 269.791,Z 650.893,A -85,B 0,C 180,E1 -17922.028,E2 -17922.028} C_VEL
LIN {X 0,Y 269.222,Z 656.587,A -85,B 0,C 180,E1 -17926.687,E2 -17926.687} C_VEL
LIN {X 0,Y 269.117,Z 658.938,A -85,B 0,C 180,E1 -17928.607,E2 -17928.607} C_VEL
LIN {X 0,Y 272.564,Z 672.933,A -85,B 0,C 180,E1 -17929.621,E2 -17929.621} C_VEL
LIN {X 0,Y 275.081,Z 684.934,A -85,B 0,C 180,E1 -17930.735,E2 -17930.735} C_VEL
LIN {X 0,Y 277.101,Z 697.573,A -85,B 0,C 180,E1 -17932.175,E2 -17932.175} C_VEL
LIN {X 0,Y 277.384,Z 700.416,A -85,B 0,C 180,E1 -17932.532,E2 -17932.532} C_VEL
LIN {X 0,Y 275.83,Z 712.084,A -85,B 0,C 180,E1 -17934.058,E2 -17934.058} C_VEL
LIN {X 0,Y 274.343,Z 721.652,A -85,B 0,C 180,E1 -17935.613,E2 -17935.613} C_VEL
LIN {X 0,Y 273.037,Z 729.789,A -85,B 0,C 180,E1 -17937.222,E2 -17937.222} C_VEL
LIN {X 0,Y 271.498,Z 738.956,A -85,B 0,C 180,E1 -17939.46,E2 -17939.46} C_VEL
LIN {X 0,Y 270.296,Z 746.476,A -85,B 0,C 180,E1 -17941.77,E2 -17941.77} C_VEL
LIN {X 0,Y 269.36,Z 752.696,A -85,B 0,C 180,E1 -17944.213,E2 -17944.213} C_VEL
LIN {X 0,Y 268.543,Z 758.032,A -85,B 0,C 180,E1 -17947.007,E2 -17947.007} C_VEL
LIN {X 0,Y 268.188,Z 760.77,A -85,B 0,C 180,E1 -17948.97,E2 -17948.97} C_VEL
LIN {X 0,Y 267.885,Z 762.816,A -85,B 0,C 180,E1 -17950.985,E2 -17950.985} C_VEL
LIN {X 0,Y 267.812,Z 764.127,A -85,B 0,C 180,E1 -17953.022,E2 -17953.022} C_VEL
LIN {X 0,Y 267.859,Z 764.661,A -85,B 0,C 180,E1 -17955.105,E2 -17955.105} C_VEL
LIN {X 0,Y 268.019,Z 764.42,A -85,B 0,C 180,E1 -17957.24,E2 -17957.24} C_VEL
LIN {X 0,Y 268.341,Z 763.349,A -85,B 0,C 180,E1 -17959.421,E2 -17959.421} C_VEL
LIN {X 0,Y 268.88,Z 761.38,A -85,B 0,C 180,E1 -17961.64,E2 -17961.64} C_VEL
LIN {X 0,Y 269.932,Z 757.453,A -85,B 0,C 180,E1 -17964.494,E2 -17964.494} C_VEL
LIN {X 0,Y 271.232,Z 752.496,A -85,B 0,C 180,E1 -17967.034,E2 -17967.034} C_VEL
LIN {X 0,Y 272.831,Z 746.335,A -85,B 0,C 180,E1 -17969.42,E2 -17969.42} C_VEL
LIN {X 0,Y 274.846,Z 738.603,A -85,B 0,C 180,E1 -17971.767,E2 -17971.767} C_VEL
LIN {X 0,Y 276.961,Z 729.991,A -85,B 0,C 180,E1 -17973.839,E2 -17973.839} C_VEL
LIN {X 0,Y 279.303,Z 720.013,A -85,B 0,C 180,E1 -17975.745,E2 -17975.745} C_VEL
LIN {X 0,Y 281.367,Z 710.126,A -85,B 0,C 180,E1 -17977.264,E2 -17977.264} C_VEL
LIN {X 0,Y 282.129,Z 705.891,A -85,B 0,C 180,E1 -17977.824,E2 -17977.824} C_VEL
LIN {X 0,Y 281.285,Z 696.915,A -85,B 0,C 180,E1 -17979.143,E2 -17979.143} C_VEL
LIN {X 0,Y 279.404,Z 686.808,A -85,B 0,C 180,E1 -17980.532,E2 -17980.532} C_VEL
LIN {X 0,Y 276.144,Z 675.366,A -85,B 0,C 180,E1 -17982.027,E2 -17982.027} C_VEL
LIN {X 0,Y 271.591,Z 663.597,A -85,B 0,C 180,E1 -17983.497,E2 -17983.497} C_VEL
LIN {X 0,Y 270.378,Z 660.513,A -85,B 0,C 180,E1 -17983.858,E2 -17983.858} C_VEL
LIN {X 0,Y 270.325,Z 660.045,A -85,B 0,C 180,E1 -17983.955,E2 -17983.955} C_VEL
LIN {X 0,Y 270.728,Z 655.431,A -85,B 0,C 180,E1 -17988.014,E2 -17988.014} C_VEL
LIN {X 0,Y 270.71,Z 652.153,A -85,B 0,C 180,E1 -17991.039,E2 -17991.039} C_VEL
LIN {X 0,Y 270.577,Z 650.786,A -85,B 0,C 180,E1 -17992.538,E2 -17992.538} C_VEL
LIN {X 0,Y 270.452,Z 650.797,A -85,B 0,C 180,E1 -17995.876,E2 -17995.876} C_VEL
LIN {X 0,Y 269.917,Z 650.864,A -85,B 0,C 180,E1 -17997.122,E2 -17997.122} C_VEL
LIN {X 0,Y 267.218,Z 651.2,A -85,B 0,C 180,E1 -17999.158,E2 -17999.158} C_VEL
LIN {X 0,Y 263.984,Z 651.603,A -85,B 0,C 180,E1 -18001.66,E2 -18001.66} C_VEL
LIN {X 0,Y 263.606,Z 651.648,A -85,B 0,C 180,E1 -18002.525,E2 -18002.525} C_VEL
LIN {X 0,Y 263.569,Z 651.652,A -85,B 0,C 180,E1 -18007.662,E2 -18007.662} C_VEL
LIN {X 0,Y 263.371,Z 651.68,A -85,B 0,C 180,E1 -18010.766,E2 -18010.766} C_VEL
LIN {X 0,Y 263.347,Z 651.683,A -85,B 0,C 180,E1 -18015.478,E2 -18015.478} C_VEL
LIN {X 0,Y 263.26,Z 651.694,A -85,B 0,C 180,E1 -18020.307,E2 -18020.307} C_VEL
LIN {X 0,Y 263.206,Z 651.7,A -85,B 0,C 180,E1 -18025.292,E2 -18025.292} C_VEL
LIN {X 0,Y 263.173,Z 651.701,A -85,B 0,C 180,E1 -18028.73,E2 -18028.73} C_VEL
LIN {X 0,Y 263.13,Z 651.71,A -85,B 0,C 180,E1 -18032.289,E2 -18032.289} C_VEL
LIN {X 0,Y 263.16,Z 651.703,A -85,B 0,C 180,E1 -18035.982,E2 -18035.982} C_VEL
LIN {X 0,Y 263.103,Z 651.71,A -85,B 0,C 180,E1 -18039.873,E2 -18039.873} C_VEL
LIN {X 0,Y 263.168,Z 651.714,A -85,B 0,C 180,E1 -18043.975,E2 -18043.975} C_VEL
LIN {X 0,Y 263.923,Z 656.106,A -85,B 0,C 180,E1 -18048.212,E2 -18048.212} C_VEL
LIN {X 0,Y 264.573,Z 659.572,A -85,B 0,C 180,E1 -18051.411,E2 -18051.411} C_VEL
LIN {X 0,Y 264.617,Z 662.843,A -85,B 0,C 180,E1 -18054.247,E2 -18054.247} C_VEL
LIN {X 0,Y 263.929,Z 667.166,A -85,B 0,C 180,E1 -18057.822,E2 -18057.822} C_VEL
LIN {X 0,Y 263.694,Z 668.806,A -85,B 0,C 180,E1 -18059.161,E2 -18059.161} C_VEL
LIN {X 0,Y 264.58,Z 672.318,A -85,B 0,C 180,E1 -18059.502,E2 -18059.502} C_VEL
LIN {X 0,Y 265.607,Z 675.117,A -85,B 0,C 180,E1 -18059.819,E2 -18059.819} C_VEL
LIN {X 0,Y 268.826,Z 685.813,A -85,B 0,C 180,E1 -18061.039,E2 -18061.039} C_VEL
LIN {X 0,Y 271.417,Z 697.444,A -85,B 0,C 180,E1 -18062.435,E2 -18062.435} C_VEL
LIN {X 0,Y 272.863,Z 708.202,A -85,B 0,C 180,E1 -18063.833,E2 -18063.833} C_VEL
LIN {X 0,Y 273.263,Z 718.581,A -85,B 0,C 180,E1 -18065.291,E2 -18065.291} C_VEL
LIN {X 0,Y 272.936,Z 727.411,A -85,B 0,C 180,E1 -18066.679,E2 -18066.679} C_VEL
LIN {X 0,Y 270.783,Z 736.996,A -85,B 0,C 180,E1 -18068.294,E2 -18068.294} C_VEL
LIN {X 0,Y 268.58,Z 745.795,A -85,B 0,C 180,E1 -18070.113,E2 -18070.113} C_VEL
LIN {X 0,Y 266.442,Z 754.462,A -85,B 0,C 180,E1 -18072.343,E2 -18072.343} C_VEL
LIN {X 0,Y 264.695,Z 761.441,A -85,B 0,C 180,E1 -18074.603,E2 -18074.603} C_VEL
LIN {X 0,Y 263.186,Z 767.052,A -85,B 0,C 180,E1 -18076.881,E2 -18076.881} C_VEL
LIN {X 0,Y 262.21,Z 771.476,A -85,B 0,C 180,E1 -18079.187,E2 -18079.187} C_VEL
LIN {X 0,Y 261.732,Z 773.824,A -85,B 0,C 180,E1 -18080.729,E2 -18080.729} C_VEL
LIN {X 0,Y 261.378,Z 775.75,A -85,B 0,C 180,E1 -18082.274,E2 -18082.274} C_VEL
LIN {X 0,Y 261.132,Z 777.922,A -85,B 0,C 180,E1 -18084.751,E2 -18084.751} C_VEL
LIN {X 0,Y 261.119,Z 779.926,A -85,B 0,C 180,E1 -18088.458,E2 -18088.458} C_VEL
LIN {X 0,Y 261.129,Z 780.515,A -85,B 0,C 180,E1 -18090.001,E2 -18090.001} C_VEL
LIN {X 0,Y 261.115,Z 780.706,A -85,B 0,C 180,E1 -18091.543,E2 -18091.543} C_VEL
LIN {X 0,Y 261.067,Z 780.459,A -85,B 0,C 180,E1 -18093.087,E2 -18093.087} C_VEL
LIN {X 0,Y 261.23,Z 778.778,A -85,B 0,C 180,E1 -18096.178,E2 -18096.178} C_VEL
LIN {X 0,Y 261.412,Z 777.348,A -85,B 0,C 180,E1 -18097.726,E2 -18097.726} C_VEL
LIN {X 0,Y 261.987,Z 774.367,A -85,B 0,C 180,E1 -18100.042,E2 -18100.042} C_VEL
LIN {X 0,Y 262.905,Z 770.372,A -85,B 0,C 180,E1 -18102.349,E2 -18102.349} C_VEL
LIN {X 0,Y 264.179,Z 765.27,A -85,B 0,C 180,E1 -18104.64,E2 -18104.64} C_VEL
LIN {X 0,Y 266.022,Z 758.926,A -85,B 0,C 180,E1 -18106.895,E2 -18106.895} C_VEL
LIN {X 0,Y 268.019,Z 750.583,A -85,B 0,C 180,E1 -18109.266,E2 -18109.266} C_VEL
LIN {X 0,Y 270.386,Z 741.378,A -85,B 0,C 180,E1 -18111.34,E2 -18111.34} C_VEL
LIN {X 0,Y 272.807,Z 731.411,A -85,B 0,C 180,E1 -18113.134,E2 -18113.134} C_VEL
LIN {X 0,Y 273.753,Z 726.795,A -85,B 0,C 180,E1 -18113.851,E2 -18113.851} C_VEL
LIN {X 0,Y 273.857,Z 717.22,A -85,B 0,C 180,E1 -18115.347,E2 -18115.347} C_VEL
LIN {X 0,Y 272.961,Z 705.916,A -85,B 0,C 180,E1 -18116.948,E2 -18116.948} C_VEL
LIN {X 0,Y 270.538,Z 693.392,A -85,B 0,C 180,E1 -18118.605,E2 -18118.605} C_VEL
LIN {X 0,Y 266.882,Z 680.835,A -85,B 0,C 180,E1 -18120.197,E2 -18120.197} C_VEL
LIN {X 0,Y 264.348,Z 674.016,A -85,B 0,C 180,E1 -18121.043,E2 -18121.043} C_VEL
LIN {X 0,Y 264.193,Z 673.005,A -85,B 0,C 180,E1 -18121.137,E2 -18121.137} C_VEL
LIN {X 0,Y 264.924,Z 669.156,A -85,B 0,C 180,E1 -18124.676,E2 -18124.676} C_VEL
LIN {X 0,Y 265.229,Z 666.249,A -85,B 0,C 180,E1 -18127.55,E2 -18127.55} C_VEL
LIN {X 0,Y 265.141,Z 664.191,A -85,B 0,C 180,E1 -18129.763,E2 -18129.763} C_VEL
LIN {X 0,Y 264.737,Z 660.928,A -85,B 0,C 180,E1 -18133.648,E2 -18133.648} C_VEL
LIN {X 0,Y 264.191,Z 657.659,A -85,B 0,C 180,E1 -18138.147,E2 -18138.147} C_VEL
LIN {X 0,Y 263.762,Z 655.188,A -85,B 0,C 180,E1 -18142.205,E2 -18142.205} C_VEL
LIN {X 0,Y 263.439,Z 653.315,A -85,B 0,C 180,E1 -18145.928,E2 -18145.928} C_VEL
LIN {X 0,Y 263.171,Z 651.908,A -85,B 0,C 180,E1 -18149.509,E2 -18149.509} C_VEL
LIN {X 0,Y 263.193,Z 651.7,A -85,B 0,C 180,E1 -18153.003,E2 -18153.003} C_VEL
LIN {X 0,Y 263.186,Z 651.698,A -85,B 0,C 180,E1 -18156.387,E2 -18156.387} C_VEL
LIN {X 0,Y 263.266,Z 651.693,A -85,B 0,C 180,E1 -18159.694,E2 -18159.694} C_VEL
LIN {X 0,Y 263.353,Z 651.682,A -85,B 0,C 180,E1 -18164.522,E2 -18164.522} C_VEL
LIN {X 0,Y 263.376,Z 651.678,A -85,B 0,C 180,E1 -18169.235,E2 -18169.235} C_VEL
LIN {X 0,Y 263.575,Z 651.651,A -85,B 0,C 180,E1 -18172.339,E2 -18172.339} C_VEL
LIN {X 0,Y 263.498,Z 652.369,A -85,B 0,C 180,E1 -18175.411,E2 -18175.411} C_VEL
LIN {X 0,Y 264.029,Z 653.49,A -85,B 0,C 180,E1 -18178.475,E2 -18178.475} C_VEL
LIN {X 0,Y 264.235,Z 654.136,A -85,B 0,C 180,E1 -18180,E2 -18180} C_VEL
LIN {X 0,Y 264.249,Z 655.665,A -85,B 0,C 180,E1 -18183.049,E2 -18183.049} C_VEL
LIN {X 0,Y 264.293,Z 657.878,A -85,B 0,C 180,E1 -18186.952,E2 -18186.952} C_VEL
LIN {X 0,Y 264.171,Z 659.908,A -85,B 0,C 180,E1 -18190.149,E2 -18190.149} C_VEL
LIN {X 0,Y 263.568,Z 662.543,A -85,B 0,C 180,E1 -18193.836,E2 -18193.836} C_VEL
LIN {X 0,Y 264.578,Z 665.604,A -85,B 0,C 180,E1 -18194.224,E2 -18194.224} C_VEL
LIN {X 0,Y 265.926,Z 668.435,A -85,B 0,C 180,E1 -18194.639,E2 -18194.639} C_VEL
LIN {X 0,Y 270.014,Z 678.793,A -85,B 0,C 180,E1 -18196.141,E2 -18196.141} C_VEL
LIN {X 0,Y 273.358,Z 690.142,A -85,B 0,C 180,E1 -18197.799,E2 -18197.799} C_VEL
LIN {X 0,Y 275.354,Z 700.44,A -85,B 0,C 180,E1 -18199.379,E2 -18199.379} C_VEL
LIN {X 0,Y 276.033,Z 707.323,A -85,B 0,C 180,E1 -18200.493,E2 -18200.493} C_VEL
LIN {X 0,Y 273.713,Z 718.657,A -85,B 0,C 180,E1 -18202.174,E2 -18202.174} C_VEL
LIN {X 0,Y 271.267,Z 728.81,A -85,B 0,C 180,E1 -18204.083,E2 -18204.083} C_VEL
LIN {X 0,Y 269.112,Z 736.82,A -85,B 0,C 180,E1 -18205.94,E2 -18205.94} C_VEL
LIN {X 0,Y 266.911,Z 744.932,A -85,B 0,C 180,E1 -18208.292,E2 -18208.292} C_VEL
LIN {X 0,Y 265.384,Z 750.229,A -85,B 0,C 180,E1 -18210.21,E2 -18210.21} C_VEL
LIN {X 0,Y 264.104,Z 754.611,A -85,B 0,C 180,E1 -18212.155,E2 -18212.155} C_VEL
LIN {X 0,Y 262.664,Z 759.72,A -85,B 0,C 180,E1 -18215.119,E2 -18215.119} C_VEL
LIN {X 0,Y 261.695,Z 763.161,A -85,B 0,C 180,E1 -18218.147,E2 -18218.147} C_VEL
LIN {X 0,Y 261.089,Z 764.988,A -85,B 0,C 180,E1 -18221.087,E2 -18221.087} C_VEL
LIN {X 0,Y 260.846,Z 765.392,A -85,B 0,C 180,E1 -18223.325,E2 -18223.325} C_VEL
LIN {X 0,Y 260.779,Z 764.963,A -85,B 0,C 180,E1 -18225.516,E2 -18225.516} C_VEL
LIN {X 0,Y 260.927,Z 763.764,A -85,B 0,C 180,E1 -18227.672,E2 -18227.672} C_VEL
LIN {X 0,Y 261.157,Z 761.846,A -85,B 0,C 180,E1 -18229.769,E2 -18229.769} C_VEL
LIN {X 0,Y 261.515,Z 759.178,A -85,B 0,C 180,E1 -18231.822,E2 -18231.822} C_VEL
LIN {X 0,Y 262.153,Z 754.79,A -85,B 0,C 180,E1 -18234.331,E2 -18234.331} C_VEL
LIN {X 0,Y 263.001,Z 748.831,A -85,B 0,C 180,E1 -18236.895,E2 -18236.895} C_VEL
LIN {X 0,Y 264.286,Z 741.429,A -85,B 0,C 180,E1 -18239.377,E2 -18239.377} C_VEL
LIN {X 0,Y 265.701,Z 733.201,A -85,B 0,C 180,E1 -18241.568,E2 -18241.568} C_VEL
LIN {X 0,Y 267.383,Z 723.292,A -85,B 0,C 180,E1 -18243.669,E2 -18243.669} C_VEL
LIN {X 0,Y 269.087,Z 712.758,A -85,B 0,C 180,E1 -18245.459,E2 -18245.459} C_VEL
LIN {X 0,Y 270.511,Z 702.357,A -85,B 0,C 180,E1 -18246.873,E2 -18246.873} C_VEL
LIN {X 0,Y 269.754,Z 695.162,A -85,B 0,C 180,E1 -18247.802,E2 -18247.802} C_VEL
LIN {X 0,Y 267.61,Z 682.973,A -85,B 0,C 180,E1 -18249.178,E2 -18249.178} C_VEL
LIN {X 0,Y 264.455,Z 669.346,A -85,B 0,C 180,E1 -18250.42,E2 -18250.42} C_VEL
LIN {X 0,Y 262.226,Z 660.592,A -85,B 0,C 180,E1 -18251.09,E2 -18251.09} C_VEL
LIN {X 0,Y 262.59,Z 657.442,A -85,B 0,C 180,E1 -18254.475,E2 -18254.475} C_VEL
LIN {X 0,Y 263.087,Z 653.179,A -85,B 0,C 180,E1 -18259.222,E2 -18259.222} C_VEL
LIN {X 0,Y 263.374,Z 651.68,A -85,B 0,C 180,E1 -18261.006,E2 -18261.006} C_VEL
LIN {X 0,Y 263.503,Z 651.66,A -85,B 0,C 180,E1 -18263.875,E2 -18263.875} C_VEL
LIN {X 0,Y 263.755,Z 651.628,A -85,B 0,C 180,E1 -18268.472,E2 -18268.472} C_VEL
LIN {X 0,Y 263.754,Z 651.626,A -85,B 0,C 180,E1 -18271.526,E2 -18271.526} C_VEL
LIN {X 0,Y 263.471,Z 651.665,A -85,B 0,C 180,E1 -18276.124,E2 -18276.124} C_VEL
LIN {X 0,Y 263.204,Z 651.699,A -85,B 0,C 180,E1 -18279.218,E2 -18279.218} C_VEL
LIN {X 0,Y 262.759,Z 651.763,A -85,B 0,C 180,E1 -18281.963,E2 -18281.963} C_VEL
LIN {X 0,Y 262.137,Z 658,A -85,B 0,C 180,E1 -18287.152,E2 -18287.152} C_VEL
LIN {X 0,Y 262.075,Z 659.054,A -85,B 0,C 180,E1 -18288.012,E2 -18288.012} C_VEL
LIN {X 0,Y 265.588,Z 673.367,A -85,B 0,C 180,E1 -18289.114,E2 -18289.114} C_VEL
LIN {X 0,Y 268.218,Z 685.807,A -85,B 0,C 180,E1 -18290.314,E2 -18290.314} C_VEL
LIN {X 0,Y 270.16,Z 698.082,A -85,B 0,C 180,E1 -18291.758,E2 -18291.758} C_VEL
LIN {X 0,Y 270.506,Z 700.896,A -85,B 0,C 180,E1 -18292.13,E2 -18292.13} C_VEL
LIN {X 0,Y 269.028,Z 712.177,A -85,B 0,C 180,E1 -18293.647,E2 -18293.647} C_VEL
LIN {X 0,Y 267.437,Z 721.986,A -85,B 0,C 180,E1 -18295.279,E2 -18295.279} C_VEL
LIN {X 0,Y 265.748,Z 731.947,A -85,B 0,C 180,E1 -18297.354,E2 -18297.354} C_VEL
LIN {X 0,Y 264.282,Z 740.441,A -85,B 0,C 180,E1 -18299.561,E2 -18299.561} C_VEL
LIN {X 0,Y 263.191,Z 747.265,A -85,B 0,C 180,E1 -18301.778,E2 -18301.778} C_VEL
LIN {X 0,Y 262.238,Z 753.256,A -85,B 0,C 180,E1 -18304.249,E2 -18304.249} C_VEL
LIN {X 0,Y 261.412,Z 758.666,A -85,B 0,C 180,E1 -18307.22,E2 -18307.22} C_VEL
LIN {X 0,Y 261.123,Z 760.65,A -85,B 0,C 180,E1 -18308.691,E2 -18308.691} C_VEL
LIN {X 0,Y 260.782,Z 762.997,A -85,B 0,C 180,E1 -18311.01,E2 -18311.01} C_VEL
LIN {X 0,Y 260.715,Z 764.392,A -85,B 0,C 180,E1 -18313.295,E2 -18313.295} C_VEL
LIN {X 0,Y 260.77,Z 764.895,A -85,B 0,C 180,E1 -18315.514,E2 -18315.514} C_VEL
LIN {X 0,Y 260.974,Z 764.565,A -85,B 0,C 180,E1 -18317.682,E2 -18317.682} C_VEL
LIN {X 0,Y 261.325,Z 763.491,A -85,B 0,C 180,E1 -18319.8,E2 -18319.8} C_VEL
LIN {X 0,Y 261.853,Z 761.705,A -85,B 0,C 180,E1 -18321.88,E2 -18321.88} C_VEL
LIN {X 0,Y 262.589,Z 759.181,A -85,B 0,C 180,E1 -18323.927,E2 -18323.927} C_VEL
LIN {X 0,Y 264.059,Z 753.928,A -85,B 0,C 180,E1 -18326.933,E2 -18326.933} C_VEL
LIN {X 0,Y 265.718,Z 748.023,A -85,B 0,C 180,E1 -18329.442,E2 -18329.442} C_VEL
LIN {X 0,Y 267.746,Z 740.813,A -85,B 0,C 180,E1 -18331.805,E2 -18331.805} C_VEL
LIN {X 0,Y 270.1,Z 732.003,A -85,B 0,C 180,E1 -18334.084,E2 -18334.084} C_VEL
LIN {X 0,Y 272.448,Z 722.512,A -85,B 0,C 180,E1 -18336.029,E2 -18336.029} C_VEL
LIN {X 0,Y 274.949,Z 711.246,A -85,B 0,C 180,E1 -18337.85,E2 -18337.85} C_VEL
LIN {X 0,Y 275.726,Z 706.57,A -85,B 0,C 180,E1 -18338.506,E2 -18338.506} C_VEL
LIN {X 0,Y 274.61,Z 695.744,A -85,B 0,C 180,E1 -18340.178,E2 -18340.178} C_VEL
LIN {X 0,Y 272.257,Z 684.687,A -85,B 0,C 180,E1 -18341.761,E2 -18341.761} C_VEL
LIN {X 0,Y 268.337,Z 672.387,A -85,B 0,C 180,E1 -18343.451,E2 -18343.451} C_VEL
LIN {X 0,Y 264.676,Z 663.576,A -85,B 0,C 180,E1 -18344.651,E2 -18344.651} C_VEL
LIN {X 0,Y 263.502,Z 660.273,A -85,B 0,C 180,E1 -18345.075,E2 -18345.075} C_VEL
LIN {X 0,Y 263.769,Z 657.385,A -85,B 0,C 180,E1 -18347.692,E2 -18347.692} C_VEL
LIN {X 0,Y 263.817,Z 654.073,A -85,B 0,C 180,E1 -18350.802,E2 -18350.802} C_VEL
LIN {X 0,Y 263.513,Z 651.665,A -85,B 0,C 180,E1 -18353.299,E2 -18353.299} C_VEL
LIN {X 0,Y 263.75,Z 651.632,A -85,B 0,C 180,E1 -18358.473,E2 -18358.473} C_VEL
LIN {X 0,Y 263.749,Z 651.633,A -85,B 0,C 180,E1 -18361.527,E2 -18361.527} C_VEL
LIN {X 0,Y 263.606,Z 651.648,A -85,B 0,C 180,E1 -18362.525,E2 -18362.525} C_VEL
LIN {X 0,Y 262.848,Z 651.745,A -85,B 0,C 180,E1 -18363.799,E2 -18363.799} C_VEL
LIN {X 0,Y 259.95,Z 652.104,A -85,B 0,C 180,E1 -18365.875,E2 -18365.875} C_VEL
LIN {X 0,Y 257.559,Z 652.401,A -85,B 0,C 180,E1 -18367.564,E2 -18367.564} C_VEL
LIN {X 0,Y 256.56,Z 652.528,A -85,B 0,C 180,E1 -18368.874,E2 -18368.874} C_VEL
LIN {X 0,Y 256.489,Z 652.533,A -85,B 0,C 180,E1 -18369.317,E2 -18369.317} C_VEL
LIN {X 0,Y 256.252,Z 652.563,A -85,B 0,C 180,E1 -18374.29,E2 -18374.29} C_VEL
LIN {X 0,Y 256.208,Z 652.572,A -85,B 0,C 180,E1 -18377.562,E2 -18377.562} C_VEL
LIN {X 0,Y 256.154,Z 652.575,A -85,B 0,C 180,E1 -18381.12,E2 -18381.12} C_VEL
LIN {X 0,Y 256.186,Z 652.575,A -85,B 0,C 180,E1 -18385.139,E2 -18385.139} C_VEL
LIN {X 0,Y 256.108,Z 652.585,A -85,B 0,C 180,E1 -18389.6,E2 -18389.6} C_VEL
LIN {X 0,Y 256.074,Z 652.585,A -85,B 0,C 180,E1 -18393.292,E2 -18393.292} C_VEL
LIN {X 0,Y 256.112,Z 652.581,A -85,B 0,C 180,E1 -18397.271,E2 -18397.271} C_VEL
LIN {X 0,Y 256.053,Z 652.591,A -85,B 0,C 180,E1 -18401.204,E2 -18401.204} C_VEL
LIN {X 0,Y 256.145,Z 652.793,A -85,B 0,C 180,E1 -18403.919,E2 -18403.919} C_VEL
LIN {X 0,Y 256.809,Z 656.538,A -85,B 0,C 180,E1 -18407.638,E2 -18407.638} C_VEL
LIN {X 0,Y 257.486,Z 660.189,A -85,B 0,C 180,E1 -18411.115,E2 -18411.115} C_VEL
LIN {X 0,Y 257.578,Z 663.513,A -85,B 0,C 180,E1 -18414.084,E2 -18414.084} C_VEL
LIN {X 0,Y 256.838,Z 668.041,A -85,B 0,C 180,E1 -18417.899,E2 -18417.899} C_VEL
LIN {X 0,Y 257.599,Z 671.179,A -85,B 0,C 180,E1 -18418.2,E2 -18418.2} C_VEL
LIN {X 0,Y 258.756,Z 674.036,A -85,B 0,C 180,E1 -18418.573,E2 -18418.573} C_VEL
LIN {X 0,Y 262.281,Z 685.074,A -85,B 0,C 180,E1 -18419.928,E2 -18419.928} C_VEL
LIN {X 0,Y 264.977,Z 697.365,A -85,B 0,C 180,E1 -18421.484,E2 -18421.484} C_VEL
LIN {X 0,Y 266.413,Z 707.831,A -85,B 0,C 180,E1 -18422.904,E2 -18422.904} C_VEL
LIN {X 0,Y 266.904,Z 718.263,A -85,B 0,C 180,E1 -18424.446,E2 -18424.446} C_VEL
LIN {X 0,Y 266.455,Z 728.194,A -85,B 0,C 180,E1 -18426.077,E2 -18426.077} C_VEL
LIN {X 0,Y 264.235,Z 737.615,A -85,B 0,C 180,E1 -18427.728,E2 -18427.728} C_VEL
LIN {X 0,Y 261.946,Z 746.281,A -85,B 0,C 180,E1 -18429.588,E2 -18429.588} C_VEL
LIN {X 0,Y 259.678,Z 754.789,A -85,B 0,C 180,E1 -18431.867,E2 -18431.867} C_VEL
LIN {X 0,Y 257.577,Z 762.636,A -85,B 0,C 180,E1 -18434.573,E2 -18434.573} C_VEL
LIN {X 0,Y 255.863,Z 768.755,A -85,B 0,C 180,E1 -18437.307,E2 -18437.307} C_VEL
LIN {X 0,Y 254.94,Z 772.743,A -85,B 0,C 180,E1 -18439.678,E2 -18439.678} C_VEL
LIN {X 0,Y 254.331,Z 775.706,A -85,B 0,C 180,E1 -18442.059,E2 -18442.059} C_VEL
LIN {X 0,Y 254.014,Z 778.144,A -85,B 0,C 180,E1 -18445.239,E2 -18445.239} C_VEL
LIN {X 0,Y 254.048,Z 779.635,A -85,B 0,C 180,E1 -18448.415,E2 -18448.415} C_VEL
LIN {X 0,Y 254.057,Z 780.255,A -85,B 0,C 180,E1 -18450.001,E2 -18450.001} C_VEL
LIN {X 0,Y 254.021,Z 780.478,A -85,B 0,C 180,E1 -18451.586,E2 -18451.586} C_VEL
LIN {X 0,Y 253.967,Z 780.289,A -85,B 0,C 180,E1 -18453.173,E2 -18453.173} C_VEL
LIN {X 0,Y 254.159,Z 778.666,A -85,B 0,C 180,E1 -18456.351,E2 -18456.351} C_VEL
LIN {X 0,Y 254.358,Z 777.266,A -85,B 0,C 180,E1 -18457.942,E2 -18457.942} C_VEL
LIN {X 0,Y 254.964,Z 774.352,A -85,B 0,C 180,E1 -18460.322,E2 -18460.322} C_VEL
LIN {X 0,Y 255.93,Z 770.441,A -85,B 0,C 180,E1 -18462.691,E2 -18462.691} C_VEL
LIN {X 0,Y 257.317,Z 765.432,A -85,B 0,C 180,E1 -18465.039,E2 -18465.039} C_VEL
LIN {X 0,Y 259.246,Z 759.183,A -85,B 0,C 180,E1 -18467.35,E2 -18467.35} C_VEL
LIN {X 0,Y 261.239,Z 751.368,A -85,B 0,C 180,E1 -18469.679,E2 -18469.679} C_VEL
LIN {X 0,Y 263.803,Z 741.893,A -85,B 0,C 180,E1 -18471.9,E2 -18471.9} C_VEL
LIN {X 0,Y 266.342,Z 732.161,A -85,B 0,C 180,E1 -18473.729,E2 -18473.729} C_VEL
LIN {X 0,Y 267.294,Z 727.669,A -85,B 0,C 180,E1 -18474.464,E2 -18474.464} C_VEL
LIN {X 0,Y 267.492,Z 718.42,A -85,B 0,C 180,E1 -18475.989,E2 -18475.989} C_VEL
LIN {X 0,Y 266.67,Z 707.117,A -85,B 0,C 180,E1 -18477.685,E2 -18477.685} C_VEL
LIN {X 0,Y 264.529,Z 695.417,A -85,B 0,C 180,E1 -18479.342,E2 -18479.342} C_VEL
LIN {X 0,Y 261.285,Z 683.884,A -85,B 0,C 180,E1 -18480.918,E2 -18480.918} C_VEL
LIN {X 0,Y 258.598,Z 676.466,A -85,B 0,C 180,E1 -18481.932,E2 -18481.932} C_VEL
LIN {X 0,Y 257.415,Z 672.95,A -85,B 0,C 180,E1 -18482.371,E2 -18482.371} C_VEL
LIN {X 0,Y 257.984,Z 669.823,A -85,B 0,C 180,E1 -18485.188,E2 -18485.188} C_VEL
LIN {X 0,Y 258.218,Z 667.224,A -85,B 0,C 180,E1 -18487.879,E2 -18487.879} C_VEL
LIN {X 0,Y 258.049,Z 664.636,A -85,B 0,C 180,E1 -18490.817,E2 -18490.817} C_VEL
LIN {X 0,Y 257.633,Z 661.476,A -85,B 0,C 180,E1 -18494.825,E2 -18494.825} C_VEL
LIN {X 0,Y 257.133,Z 658.651,A -85,B 0,C 180,E1 -18499.007,E2 -18499.007} C_VEL
LIN {X 0,Y 256.778,Z 656.372,A -85,B 0,C 180,E1 -18502.977,E2 -18502.977} C_VEL
LIN {X 0,Y 256.436,Z 654.626,A -85,B 0,C 180,E1 -18506.761,E2 -18506.761} C_VEL
LIN {X 0,Y 256.215,Z 653.305,A -85,B 0,C 180,E1 -18510.413,E2 -18510.413} C_VEL
LIN {X 0,Y 256.138,Z 652.576,A -85,B 0,C 180,E1 -18513.959,E2 -18513.959} C_VEL
LIN {X 0,Y 256.102,Z 652.585,A -85,B 0,C 180,E1 -18517.407,E2 -18517.407} C_VEL
LIN {X 0,Y 256.189,Z 652.575,A -85,B 0,C 180,E1 -18520.78,E2 -18520.78} C_VEL
LIN {X 0,Y 256.302,Z 652.56,A -85,B 0,C 180,E1 -18524.085,E2 -18524.085} C_VEL
LIN {X 0,Y 256.312,Z 652.559,A -85,B 0,C 180,E1 -18528.934,E2 -18528.934} C_VEL
LIN {X 0,Y 256.499,Z 652.532,A -85,B 0,C 180,E1 -18530.538,E2 -18530.538} C_VEL
LIN {X 0,Y 256.595,Z 653.351,A -85,B 0,C 180,E1 -18533.71,E2 -18533.71} C_VEL
LIN {X 0,Y 257.095,Z 654.977,A -85,B 0,C 180,E1 -18538.434,E2 -18538.434} C_VEL
LIN {X 0,Y 257.294,Z 655.616,A -85,B 0,C 180,E1 -18540,E2 -18540} C_VEL
LIN {X 0,Y 257.297,Z 657.129,A -85,B 0,C 180,E1 -18543.132,E2 -18543.132} C_VEL
LIN {X 0,Y 257.316,Z 659.216,A -85,B 0,C 180,E1 -18546.944,E2 -18546.944} C_VEL
LIN {X 0,Y 257.143,Z 661.289,A -85,B 0,C 180,E1 -18550.288,E2 -18550.288} C_VEL
LIN {X 0,Y 256.731,Z 662.832,A -85,B 0,C 180,E1 -18552.55,E2 -18552.55} C_VEL
LIN {X 0,Y 257.874,Z 666.108,A -85,B 0,C 180,E1 -18553.006,E2 -18553.006} C_VEL
LIN {X 0,Y 258.96,Z 668.254,A -85,B 0,C 180,E1 -18553.362,E2 -18553.362} C_VEL
LIN {X 0,Y 263.022,Z 678.04,A -85,B 0,C 180,E1 -18554.903,E2 -18554.903} C_VEL
LIN {X 0,Y 266.247,Z 688.163,A -85,B 0,C 180,E1 -18556.485,E2 -18556.485} C_VEL
LIN {X 0,Y 268.663,Z 699.503,A -85,B 0,C 180,E1 -18558.295,E2 -18558.295} C_VEL
LIN {X 0,Y 269.672,Z 708.421,A -85,B 0,C 180,E1 -18559.804,E2 -18559.804} C_VEL
LIN {X 0,Y 268.387,Z 715.291,A -85,B 0,C 180,E1 -18560.843,E2 -18560.843} C_VEL
LIN {X 0,Y 266.002,Z 725.112,A -85,B 0,C 180,E1 -18562.577,E2 -18562.577} C_VEL
LIN {X 0,Y 263.616,Z 733.769,A -85,B 0,C 180,E1 -18564.457,E2 -18564.457} C_VEL
LIN {X 0,Y 261.185,Z 742.181,A -85,B 0,C 180,E1 -18566.73,E2 -18566.73} C_VEL
LIN {X 0,Y 258.979,Z 749.43,A -85,B 0,C 180,E1 -18569.24,E2 -18569.24} C_VEL
LIN {X 0,Y 257.06,Z 755.672,A -85,B 0,C 180,E1 -18572.054,E2 -18572.054} C_VEL
LIN {X 0,Y 255.827,Z 759.696,A -85,B 0,C 180,E1 -18574.497,E2 -18574.497} C_VEL
LIN {X 0,Y 254.823,Z 762.987,A -85,B 0,C 180,E1 -18577.356,E2 -18577.356} C_VEL
LIN {X 0,Y 254.27,Z 764.584,A -85,B 0,C 180,E1 -18579.473,E2 -18579.473} C_VEL
LIN {X 0,Y 253.914,Z 765.432,A -85,B 0,C 180,E1 -18581.64,E2 -18581.64} C_VEL
LIN {X 0,Y 253.709,Z 765.537,A -85,B 0,C 180,E1 -18583.926,E2 -18583.926} C_VEL
LIN {X 0,Y 253.718,Z 764.846,A -85,B 0,C 180,E1 -18586.171,E2 -18586.171} C_VEL
LIN {X 0,Y 253.917,Z 763.394,A -85,B 0,C 180,E1 -18588.372,E2 -18588.372} C_VEL
LIN {X 0,Y 254.203,Z 760.929,A -85,B 0,C 180,E1 -18590.726,E2 -18590.726} C_VEL
LIN {X 0,Y 254.692,Z 757.356,A -85,B 0,C 180,E1 -18593.152,E2 -18593.152} C_VEL
LIN {X 0,Y 255.415,Z 752.487,A -85,B 0,C 180,E1 -18595.638,E2 -18595.638} C_VEL
LIN {X 0,Y 256.477,Z 746.107,A -85,B 0,C 180,E1 -18598.154,E2 -18598.154} C_VEL
LIN {X 0,Y 257.928,Z 737.967,A -85,B 0,C 180,E1 -18600.685,E2 -18600.685} C_VEL
LIN {X 0,Y 259.549,Z 728.737,A -85,B 0,C 180,E1 -18602.946,E2 -18602.946} C_VEL
LIN {X 0,Y 261.215,Z 719.244,A -85,B 0,C 180,E1 -18604.813,E2 -18604.813} C_VEL
LIN {X 0,Y 262.965,Z 708.124,A -85,B 0,C 180,E1 -18606.574,E2 -18606.574} C_VEL
LIN {X 0,Y 263.677,Z 702.936,A -85,B 0,C 180,E1 -18607.264,E2 -18607.264} C_VEL
LIN {X 0,Y 262.38,Z 692.84,A -85,B 0,C 180,E1 -18608.595,E2 -18608.595} C_VEL
LIN {X 0,Y 260.272,Z 681.572,A -85,B 0,C 180,E1 -18609.861,E2 -18609.861} C_VEL
LIN {X 0,Y 257.06,Z 668.193,A -85,B 0,C 180,E1 -18611.106,E2 -18611.106} C_VEL
LIN {X 0,Y 255.188,Z 660.773,A -85,B 0,C 180,E1 -18611.691,E2 -18611.691} C_VEL
LIN {X 0,Y 255.618,Z 657.193,A -85,B 0,C 180,E1 -18615.673,E2 -18615.673} C_VEL
LIN {X 0,Y 256.326,Z 652.623,A -85,B 0,C 180,E1 -18620.897,E2 -18620.897} C_VEL
LIN {X 0,Y 256.471,Z 652.536,A -85,B 0,C 180,E1 -18623.706,E2 -18623.706} C_VEL
LIN {X 0,Y 256.717,Z 652.505,A -85,B 0,C 180,E1 -18628.431,E2 -18628.431} C_VEL
LIN {X 0,Y 256.717,Z 652.503,A -85,B 0,C 180,E1 -18631.568,E2 -18631.568} C_VEL
LIN {X 0,Y 256.433,Z 652.542,A -85,B 0,C 180,E1 -18636.293,E2 -18636.293} C_VEL
LIN {X 0,Y 256.113,Z 652.582,A -85,B 0,C 180,E1 -18639.476,E2 -18639.476} C_VEL
LIN {X 0,Y 255.727,Z 652.665,A -85,B 0,C 180,E1 -18641.894,E2 -18641.894} C_VEL
LIN {X 0,Y 255.129,Z 658.486,A -85,B 0,C 180,E1 -18646.812,E2 -18646.812} C_VEL
LIN {X 0,Y 255.072,Z 659.228,A -85,B 0,C 180,E1 -18647.435,E2 -18647.435} C_VEL
LIN {X 0,Y 258.749,Z 674.054,A -85,B 0,C 180,E1 -18648.611,E2 -18648.611} C_VEL
LIN {X 0,Y 261.27,Z 686.419,A -85,B 0,C 180,E1 -18649.852,E2 -18649.852} C_VEL
LIN {X 0,Y 263.207,Z 698.563,A -85,B 0,C 180,E1 -18651.333,E2 -18651.333} C_VEL
LIN {X 0,Y 263.539,Z 702.903,A -85,B 0,C 180,E1 -18651.921,E2 -18651.921} C_VEL
LIN {X 0,Y 261.882,Z 714.199,A -85,B 0,C 180,E1 -18653.527,E2 -18653.527} C_VEL
LIN {X 0,Y 260.123,Z 724.64,A -85,B 0,C 180,E1 -18655.405,E2 -18655.405} C_VEL
LIN {X 0,Y 258.449,Z 734.154,A -85,B 0,C 180,E1 -18657.533,E2 -18657.533} C_VEL
LIN {X 0,Y 256.951,Z 742.656,A -85,B 0,C 180,E1 -18659.944,E2 -18659.944} C_VEL
LIN {X 0,Y 255.781,Z 749.76,A -85,B 0,C 180,E1 -18662.488,E2 -18662.488} C_VEL
LIN {X 0,Y 254.767,Z 755.927,A -85,B 0,C 180,E1 -18665.401,E2 -18665.401} C_VEL
LIN {X 0,Y 254.114,Z 760.41,A -85,B 0,C 180,E1 -18668.317,E2 -18668.317} C_VEL
LIN {X 0,Y 253.878,Z 761.821,A -85,B 0,C 180,E1 -18669.545,E2 -18669.545} C_VEL
LIN {X 0,Y 253.646,Z 763.639,A -85,B 0,C 180,E1 -18671.68,E2 -18671.68} C_VEL
LIN {X 0,Y 253.616,Z 764.751,A -85,B 0,C 180,E1 -18673.905,E2 -18673.905} C_VEL
LIN {X 0,Y 253.713,Z 765.081,A -85,B 0,C 180,E1 -18676.17,E2 -18676.17} C_VEL
LIN {X 0,Y 253.979,Z 764.626,A -85,B 0,C 180,E1 -18678.385,E2 -18678.385} C_VEL
LIN {X 0,Y 254.424,Z 763.322,A -85,B 0,C 180,E1 -18680.663,E2 -18680.663} C_VEL
LIN {X 0,Y 255.502,Z 759.975,A -85,B 0,C 180,E1 -18683.901,E2 -18683.901} C_VEL
LIN {X 0,Y 256.886,Z 755.371,A -85,B 0,C 180,E1 -18686.827,E2 -18686.827} C_VEL
LIN {X 0,Y 258.727,Z 749.291,A -85,B 0,C 180,E1 -18689.594,E2 -18689.594} C_VEL
LIN {X 0,Y 260.567,Z 743.128,A -85,B 0,C 180,E1 -18691.782,E2 -18691.782} C_VEL
LIN {X 0,Y 262.558,Z 736.154,A -85,B 0,C 180,E1 -18693.79,E2 -18693.79} C_VEL
LIN {X 0,Y 265.09,Z 726.843,A -85,B 0,C 180,E1 -18695.945,E2 -18695.945} C_VEL
LIN {X 0,Y 267.651,Z 716.435,A -85,B 0,C 180,E1 -18697.85,E2 -18697.85} C_VEL
LIN {X 0,Y 269.309,Z 708.963,A -85,B 0,C 180,E1 -18698.972,E2 -18698.972} C_VEL
LIN {X 0,Y 268.874,Z 701.408,A -85,B 0,C 180,E1 -18700.216,E2 -18700.216} C_VEL
LIN {X 0,Y 267.009,Z 690.398,A -85,B 0,C 180,E1 -18701.927,E2 -18701.927} C_VEL
LIN {X 0,Y 264.171,Z 679.75,A -85,B 0,C 180,E1 -18703.517,E2 -18703.517} C_VEL
LIN {X 0,Y 260.008,Z 668.335,A -85,B 0,C 180,E1 -18705.171,E2 -18705.171} C_VEL
LIN {X 0,Y 257.791,Z 663.612,A -85,B 0,C 180,E1 -18705.897,E2 -18705.897} C_VEL
LIN {X 0,Y 256.7,Z 660.47,A -85,B 0,C 180,E1 -18706.341,E2 -18706.341} C_VEL
LIN {X 0,Y 256.944,Z 656.665,A -85,B 0,C 180,E1 -18709.952,E2 -18709.952} C_VEL
LIN {X 0,Y 256.812,Z 654.5,A -85,B 0,C 180,E1 -18712.135,E2 -18712.135} C_VEL
LIN {X 0,Y 256.404,Z 652.55,A -85,B 0,C 180,E1 -18714.298,E2 -18714.298} C_VEL
LIN {X 0,Y 256.712,Z 652.509,A -85,B 0,C 180,E1 -18718.431,E2 -18718.431} C_VEL
LIN {X 0,Y 256.712,Z 652.509,A -85,B 0,C 180,E1 -18721.569,E2 -18721.569} C_VEL
LIN {X 0,Y 256.537,Z 652.529,A -85,B 0,C 180,E1 -18727.873,E2 -18727.873} C_VEL
LIN {X 0,Y 256.489,Z 652.533,A -85,B 0,C 180,E1 -18729.317,E2 -18729.317} C_VEL
LIN {X 0,Y 256.176,Z 652.576,A -85,B 0,C 180,E1 -18730.192,E2 -18730.192} C_VEL
LIN {X 0,Y 254.779,Z 652.752,A -85,B 0,C 180,E1 -18731.482,E2 -18731.482} C_VEL
LIN {X 0,Y 250.309,Z 653.303,A -85,B 0,C 180,E1 -18734.485,E2 -18734.485} C_VEL
LIN {X 0,Y 249.285,Z 653.433,A -85,B 0,C 180,E1 -18735.833,E2 -18735.833} C_VEL
LIN {X 0,Y 249.232,Z 653.437,A -85,B 0,C 180,E1 -18736.29,E2 -18736.29} C_VEL
LIN {X 0,Y 249.092,Z 653.454,A -85,B 0,C 180,E1 -18741.399,E2 -18741.399} C_VEL
LIN {X 0,Y 249.128,Z 653.452,A -85,B 0,C 180,E1 -18745.483,E2 -18745.483} C_VEL
LIN {X 0,Y 249.078,Z 653.457,A -85,B 0,C 180,E1 -18748.993,E2 -18748.993} C_VEL
LIN {X 0,Y 249.031,Z 653.466,A -85,B 0,C 180,E1 -18752.426,E2 -18752.426} C_VEL
LIN {X 0,Y 249.055,Z 653.462,A -85,B 0,C 180,E1 -18756.341,E2 -18756.341} C_VEL
LIN {X 0,Y 249.004,Z 653.467,A -85,B 0,C 180,E1 -18760.479,E2 -18760.479} C_VEL
LIN {X 0,Y 249.062,Z 653.481,A -85,B 0,C 180,E1 -18763.475,E2 -18763.475} C_VEL
LIN {X 0,Y 249.771,Z 657.439,A -85,B 0,C 180,E1 -18767.523,E2 -18767.523} C_VEL
LIN {X 0,Y 250.502,Z 661.826,A -85,B 0,C 180,E1 -18771.773,E2 -18771.773} C_VEL
LIN {X 0,Y 250.462,Z 664.784,A -85,B 0,C 180,E1 -18774.464,E2 -18774.464} C_VEL
LIN {X 0,Y 250.085,Z 667.088,A -85,B 0,C 180,E1 -18776.488,E2 -18776.488} C_VEL
LIN {X 0,Y 250.906,Z 670.489,A -85,B 0,C 180,E1 -18776.848,E2 -18776.848} C_VEL
LIN {X 0,Y 252.043,Z 673.22,A -85,B 0,C 180,E1 -18777.234,E2 -18777.234} C_VEL
LIN {X 0,Y 255.196,Z 682.73,A -85,B 0,C 180,E1 -18778.497,E2 -18778.497} C_VEL
LIN {X 0,Y 258.011,Z 694.05,A -85,B 0,C 180,E1 -18780.021,E2 -18780.021} C_VEL
LIN {X 0,Y 259.806,Z 705.306,A -85,B 0,C 180,E1 -18781.611,E2 -18781.611} C_VEL
LIN {X 0,Y 260.563,Z 716.652,A -85,B 0,C 180,E1 -18783.333,E2 -18783.333} C_VEL
LIN {X 0,Y 260.221,Z 726.861,A -85,B 0,C 180,E1 -18785.04,E2 -18785.04} C_VEL
LIN {X 0,Y 259.276,Z 732.335,A -85,B 0,C 180,E1 -18786.01,E2 -18786.01} C_VEL
LIN {X 0,Y 256.741,Z 741.854,A -85,B 0,C 180,E1 -18787.891,E2 -18787.891} C_VEL
LIN {X 0,Y 254.107,Z 750.904,A -85,B 0,C 180,E1 -18790.113,E2 -18790.113} C_VEL
LIN {X 0,Y 251.966,Z 758.663,A -85,B 0,C 180,E1 -18792.552,E2 -18792.552} C_VEL
LIN {X 0,Y 249.82,Z 765.641,A -85,B 0,C 180,E1 -18795.334,E2 -18795.334} C_VEL
LIN {X 0,Y 248.556,Z 770.281,A -85,B 0,C 180,E1 -18797.757,E2 -18797.757} C_VEL
LIN {X 0,Y 247.686,Z 773.832,A -85,B 0,C 180,E1 -18800.199,E2 -18800.199} C_VEL
LIN {X 0,Y 247.281,Z 775.646,A -85,B 0,C 180,E1 -18801.831,E2 -18801.831} C_VEL
LIN {X 0,Y 246.922,Z 778.022,A -85,B 0,C 180,E1 -18805.102,E2 -18805.102} C_VEL
LIN {X 0,Y 246.986,Z 779.995,A -85,B 0,C 180,E1 -18810.001,E2 -18810.001} C_VEL
LIN {X 0,Y 246.928,Z 780.248,A -85,B 0,C 180,E1 -18811.632,E2 -18811.632} C_VEL
LIN {X 0,Y 246.871,Z 780.106,A -85,B 0,C 180,E1 -18813.265,E2 -18813.265} C_VEL
LIN {X 0,Y 246.945,Z 779.447,A -85,B 0,C 180,E1 -18815.064,E2 -18815.064} C_VEL
LIN {X 0,Y 247.303,Z 777.202,A -85,B 0,C 180,E1 -18818.17,E2 -18818.17} C_VEL
LIN {X 0,Y 247.948,Z 774.364,A -85,B 0,C 180,E1 -18820.617,E2 -18820.617} C_VEL
LIN {X 0,Y 248.968,Z 770.526,A -85,B 0,C 180,E1 -18823.052,E2 -18823.052} C_VEL
LIN {X 0,Y 250.471,Z 765.595,A -85,B 0,C 180,E1 -18825.46,E2 -18825.46} C_VEL
LIN {X 0,Y 252.466,Z 759.434,A -85,B 0,C 180,E1 -18827.832,E2 -18827.832} C_VEL
LIN {X 0,Y 254.468,Z 752.169,A -85,B 0,C 180,E1 -18830.111,E2 -18830.111} C_VEL
LIN {X 0,Y 256.75,Z 744.254,A -85,B 0,C 180,E1 -18832.11,E2 -18832.11} C_VEL
LIN {X 0,Y 259.675,Z 733.982,A -85,B 0,C 180,E1 -18834.165,E2 -18834.165} C_VEL
LIN {X 0,Y 260.872,Z 728.551,A -85,B 0,C 180,E1 -18835.108,E2 -18835.108} C_VEL
LIN {X 0,Y 261.146,Z 719.53,A -85,B 0,C 180,E1 -18836.669,E2 -18836.669} C_VEL
LIN {X 0,Y 260.414,Z 708.372,A -85,B 0,C 180,E1 -18838.459,E2 -18838.459} C_VEL
LIN {X 0,Y 258.391,Z 696.525,A -85,B 0,C 180,E1 -18840.243,E2 -18840.243} C_VEL
LIN {X 0,Y 254.611,Z 683.411,A -85,B 0,C 180,E1 -18842.184,E2 -18842.184} C_VEL
LIN {X 0,Y 252.028,Z 676.49,A -85,B 0,C 180,E1 -18843.22,E2 -18843.22} C_VEL
LIN {X 0,Y 250.791,Z 673.37,A -85,B 0,C 180,E1 -18843.679,E2 -18843.679} C_VEL
LIN {X 0,Y 250.663,Z 672.395,A -85,B 0,C 180,E1 -18843.827,E2 -18843.827} C_VEL
LIN {X 0,Y 251.057,Z 670.258,A -85,B 0,C 180,E1 -18846.006,E2 -18846.006} C_VEL
LIN {X 0,Y 251.235,Z 668.001,A -85,B 0,C 180,E1 -18848.439,E2 -18848.439} C_VEL
LIN {X 0,Y 250.932,Z 664.87,A -85,B 0,C 180,E1 -18852.236,E2 -18852.236} C_VEL
LIN {X 0,Y 250.599,Z 662.479,A -85,B 0,C 180,E1 -18855.483,E2 -18855.483} C_VEL
LIN {X 0,Y 250.121,Z 659.758,A -85,B 0,C 180,E1 -18859.739,E2 -18859.739} C_VEL
LIN {X 0,Y 249.768,Z 657.598,A -85,B 0,C 180,E1 -18863.779,E2 -18863.779} C_VEL
LIN {X 0,Y 249.465,Z 655.926,A -85,B 0,C 180,E1 -18867.691,E2 -18867.691} C_VEL
LIN {X 0,Y 249.309,Z 654.706,A -85,B 0,C 180,E1 -18871.365,E2 -18871.365} C_VEL
LIN {X 0,Y 249.203,Z 653.867,A -85,B 0,C 180,E1 -18874.974,E2 -18874.974} C_VEL
LIN {X 0,Y 249.098,Z 653.457,A -85,B 0,C 180,E1 -18878.601,E2 -18878.601} C_VEL
LIN {X 0,Y 249.245,Z 653.439,A -85,B 0,C 180,E1 -18883.622,E2 -18883.622} C_VEL
LIN {X 0,Y 249.27,Z 653.564,A -85,B 0,C 180,E1 -18886.965,E2 -18886.965} C_VEL
LIN {X 0,Y 249.545,Z 654.09,A -85,B 0,C 180,E1 -18890.306,E2 -18890.306} C_VEL
LIN {X 0,Y 249.688,Z 654.886,A -85,B 0,C 180,E1 -18893.535,E2 -18893.535} C_VEL
LIN {X 0,Y 250.17,Z 656.466,A -85,B 0,C 180,E1 -18898.39,E2 -18898.39} C_VEL
LIN {X 0,Y 250.362,Z 657.099,A -85,B 0,C 180,E1 -18900,E2 -18900} C_VEL
LIN {X 0,Y 250.338,Z 658.6,A -85,B 0,C 180,E1 -18903.219,E2 -18903.219} C_VEL
LIN {X 0,Y 250.345,Z 660.565,A -85,B 0,C 180,E1 -18906.923,E2 -18906.923} C_VEL
LIN {X 0,Y 250.11,Z 662.665,A -85,B 0,C 180,E1 -18910.425,E2 -18910.425} C_VEL
LIN {X 0,Y 249.96,Z 663.163,A -85,B 0,C 180,E1 -18911.178,E2 -18911.178} C_VEL
LIN {X 0,Y 250.908,Z 666.089,A -85,B 0,C 180,E1 -18911.588,E2 -18911.588} C_VEL
LIN {X 0,Y 252.293,Z 668.668,A -85,B 0,C 180,E1 -18912.062,E2 -18912.062} C_VEL
LIN {X 0,Y 256.324,Z 678.075,A -85,B 0,C 180,E1 -18913.679,E2 -18913.679} C_VEL
LIN {X 0,Y 260.153,Z 689.977,A -85,B 0,C 180,E1 -18915.673,E2 -18915.673} C_VEL
LIN {X 0,Y 262.382,Z 700.929,A -85,B 0,C 180,E1 -18917.538,E2 -18917.538} C_VEL
LIN {X 0,Y 263.372,Z 710.627,A -85,B 0,C 180,E1 -18919.283,E2 -18919.283} C_VEL
LIN {X 0,Y 260.666,Z 721.905,A -85,B 0,C 180,E1 -18921.138,E2 -18921.138} C_VEL
LIN {X 0,Y 258.035,Z 731.409,A -85,B 0,C 180,E1 -18923.096,E2 -18923.096} C_VEL
LIN {X 0,Y 255.239,Z 740.602,A -85,B 0,C 180,E1 -18925.509,E2 -18925.509} C_VEL
LIN {X 0,Y 253.1,Z 747.366,A -85,B 0,C 180,E1 -18927.747,E2 -18927.747} C_VEL
LIN {X 0,Y 251.104,Z 753.388,A -85,B 0,C 180,E1 -18930.251,E2 -18930.251} C_VEL
LIN {X 0,Y 249.274,Z 758.926,A -85,B 0,C 180,E1 -18933.351,E2 -18933.351} C_VEL
LIN {X 0,Y 248.581,Z 761.069,A -85,B 0,C 180,E1 -18934.924,E2 -18934.924} C_VEL
LIN {X 0,Y 247.708,Z 763.588,A -85,B 0,C 180,E1 -18937.399,E2 -18937.399} C_VEL
LIN {X 0,Y 247.105,Z 765.129,A -85,B 0,C 180,E1 -18939.832,E2 -18939.832} C_VEL
LIN {X 0,Y 246.664,Z 765.829,A -85,B 0,C 180,E1 -18943.143,E2 -18943.143} C_VEL
LIN {X 0,Y 246.587,Z 765.33,A -85,B 0,C 180,E1 -18945.441,E2 -18945.441} C_VEL
LIN {X 0,Y 246.748,Z 764.004,A -85,B 0,C 180,E1 -18947.778,E2 -18947.778} C_VEL
LIN {X 0,Y 247.022,Z 761.754,A -85,B 0,C 180,E1 -18950.191,E2 -18950.191} C_VEL
LIN {X 0,Y 247.656,Z 757.242,A -85,B 0,C 180,E1 -18953.42,E2 -18953.42} C_VEL
LIN {X 0,Y 248.461,Z 752.12,A -85,B 0,C 180,E1 -18956.037,E2 -18956.037} C_VEL
LIN {X 0,Y 249.633,Z 745.367,A -85,B 0,C 180,E1 -18958.706,E2 -18958.706} C_VEL
LIN {X 0,Y 250.982,Z 738.052,A -85,B 0,C 180,E1 -18961.003,E2 -18961.003} C_VEL
LIN {X 0,Y 252.651,Z 728.874,A -85,B 0,C 180,E1 -18963.304,E2 -18963.304} C_VEL
LIN {X 0,Y 254.426,Z 718.913,A -85,B 0,C 180,E1 -18965.304,E2 -18965.304} C_VEL
LIN {X 0,Y 256.138,Z 708.517,A -85,B 0,C 180,E1 -18966.983,E2 -18966.983} C_VEL
LIN {X 0,Y 256.826,Z 703.416,A -85,B 0,C 180,E1 -18967.685,E2 -18967.685} C_VEL
LIN {X 0,Y 255.209,Z 692.017,A -85,B 0,C 180,E1 -18969.233,E2 -18969.233} C_VEL
LIN {X 0,Y 253.035,Z 680.724,A -85,B 0,C 180,E1 -18970.53,E2 -18970.53} C_VEL
LIN {X 0,Y 249.918,Z 667.557,A -85,B 0,C 180,E1 -18971.768,E2 -18971.768} C_VEL
LIN {X 0,Y 248.176,Z 661.016,A -85,B 0,C 180,E1 -18972.276,E2 -18972.276} C_VEL
LIN {X 0,Y 248.528,Z 658.382,A -85,B 0,C 180,E1 -18975.255,E2 -18975.255} C_VEL
LIN {X 0,Y 249.252,Z 653.717,A -85,B 0,C 180,E1 -18980.708,E2 -18980.708} C_VEL
LIN {X 0,Y 249.385,Z 653.418,A -85,B 0,C 180,E1 -18981.899,E2 -18981.899} C_VEL
LIN {X 0,Y 249.297,Z 653.431,A -85,B 0,C 180,E1 -18985.148,E2 -18985.148} C_VEL
LIN {X 0,Y 249.679,Z 653.381,A -85,B 0,C 180,E1 -18988.386,E2 -18988.386} C_VEL
LIN {X 0,Y 249.679,Z 653.379,A -85,B 0,C 180,E1 -18991.612,E2 -18991.612} C_VEL
LIN {X 0,Y 249.393,Z 653.42,A -85,B 0,C 180,E1 -18996.472,E2 -18996.472} C_VEL
LIN {X 0,Y 249.022,Z 653.464,A -85,B 0,C 180,E1 -18999.748,E2 -18999.748} C_VEL
LIN {X 0,Y 248.709,Z 653.558,A -85,B 0,C 180,E1 -19001.821,E2 -19001.821} C_VEL
LIN {X 0,Y 248.067,Z 659.371,A -85,B 0,C 180,E1 -19006.828,E2 -19006.828} C_VEL
LIN {X 0,Y 251.675,Z 673.78,A -85,B 0,C 180,E1 -19007.993,E2 -19007.993} C_VEL
LIN {X 0,Y 254.099,Z 685.35,A -85,B 0,C 180,E1 -19009.174,E2 -19009.174} C_VEL
LIN {X 0,Y 256.104,Z 697.559,A -85,B 0,C 180,E1 -19010.689,E2 -19010.689} C_VEL
LIN {X 0,Y 256.742,Z 702.989,A -85,B 0,C 180,E1 -19011.454,E2 -19011.454} C_VEL
LIN {X 0,Y 255.028,Z 714.435,A -85,B 0,C 180,E1 -19013.122,E2 -19013.122} C_VEL
LIN {X 0,Y 253.236,Z 724.814,A -85,B 0,C 180,E1 -19015.038,E2 -19015.038} C_VEL
LIN {X 0,Y 251.595,Z 733.813,A -85,B 0,C 180,E1 -19017.092,E2 -19017.092} C_VEL
LIN {X 0,Y 250.104,Z 741.971,A -85,B 0,C 180,E1 -19019.412,E2 -19019.412} C_VEL
LIN {X 0,Y 248.824,Z 749.363,A -85,B 0,C 180,E1 -19022.075,E2 -19022.075} C_VEL
LIN {X 0,Y 247.892,Z 755.036,A -85,B 0,C 180,E1 -19024.696,E2 -19024.696} C_VEL
LIN {X 0,Y 247.191,Z 759.208,A -85,B 0,C 180,E1 -19027.242,E2 -19027.242} C_VEL
LIN {X 0,Y 246.745,Z 762.179,A -85,B 0,C 180,E1 -19029.732,E2 -19029.732} C_VEL
LIN {X 0,Y 246.524,Z 764.113,A -85,B 0,C 180,E1 -19032.164,E2 -19032.164} C_VEL
LIN {X 0,Y 246.561,Z 765.249,A -85,B 0,C 180,E1 -19035.446,E2 -19035.446} C_VEL
LIN {X 0,Y 246.783,Z 765.093,A -85,B 0,C 180,E1 -19037.768,E2 -19037.768} C_VEL
LIN {X 0,Y 247.197,Z 764.108,A -85,B 0,C 180,E1 -19040.14,E2 -19040.14} C_VEL
LIN {X 0,Y 247.877,Z 762.23,A -85,B 0,C 180,E1 -19042.548,E2 -19042.548} C_VEL
LIN {X 0,Y 249.168,Z 758.375,A -85,B 0,C 180,E1 -19045.659,E2 -19045.659} C_VEL
LIN {X 0,Y 250.672,Z 753.773,A -85,B 0,C 180,E1 -19048.285,E2 -19048.285} C_VEL
LIN {X 0,Y 252.624,Z 747.732,A -85,B 0,C 180,E1 -19050.892,E2 -19050.892} C_VEL
LIN {X 0,Y 255.071,Z 739.923,A -85,B 0,C 180,E1 -19053.5,E2 -19053.5} C_VEL
LIN {X 0,Y 257.398,Z 732.093,A -85,B 0,C 180,E1 -19055.578,E2 -19055.578} C_VEL
LIN {X 0,Y 259.88,Z 723.293,A -85,B 0,C 180,E1 -19057.453,E2 -19057.453} C_VEL
LIN {X 0,Y 262.421,Z 712.998,A -85,B 0,C 180,E1 -19059.216,E2 -19059.216} C_VEL
LIN {X 0,Y 263.029,Z 710.008,A -85,B 0,C 180,E1 -19059.674,E2 -19059.674} C_VEL
LIN {X 0,Y 262.383,Z 700.886,A -85,B 0,C 180,E1 -19061.251,E2 -19061.251} C_VEL
LIN {X 0,Y 260.46,Z 690.249,A -85,B 0,C 180,E1 -19063.005,E2 -19063.005} C_VEL
LIN {X 0,Y 257.732,Z 680.239,A -85,B 0,C 180,E1 -19064.581,E2 -19064.581} C_VEL
LIN {X 0,Y 253.32,Z 668.541,A -85,B 0,C 180,E1 -19066.442,E2 -19066.442} C_VEL
LIN {X 0,Y 251.51,Z 664.605,A -85,B 0,C 180,E1 -19067.083,E2 -19067.083} C_VEL
LIN {X 0,Y 250.081,Z 661.454,A -85,B 0,C 180,E1 -19067.575,E2 -19067.575} C_VEL
LIN {X 0,Y 249.926,Z 660.645,A -85,B 0,C 180,E1 -19067.722,E2 -19067.722} C_VEL
LIN {X 0,Y 250.046,Z 658.072,A -85,B 0,C 180,E1 -19070.291,E2 -19070.291} C_VEL
LIN {X 0,Y 249.719,Z 655.042,A -85,B 0,C 180,E1 -19073.536,E2 -19073.536} C_VEL
LIN {X 0,Y 249.317,Z 653.432,A -85,B 0,C 180,E1 -19075.554,E2 -19075.554} C_VEL
LIN {X 0,Y 249.674,Z 653.386,A -85,B 0,C 180,E1 -19078.387,E2 -19078.387} C_VEL
LIN {X 0,Y 249.674,Z 653.385,A -85,B 0,C 180,E1 -19081.613,E2 -19081.613} C_VEL
LIN {X 0,Y 249.459,Z 653.413,A -85,B 0,C 180,E1 -19086.47,E2 -19086.47} C_VEL
LIN {X 0,Y 249.421,Z 653.414,A -85,B 0,C 180,E1 -19089.733,E2 -19089.733} C_VEL
LIN {X 0,Y 249.202,Z 653.442,A -85,B 0,C 180,E1 -19094.704,E2 -19094.704} C_VEL
LIN {X 0,Y 249.232,Z 653.437,A -85,B 0,C 180,E1 -19096.29,E2 -19096.29} C_VEL
LIN {X 0,Y 248.61,Z 653.52,A -85,B 0,C 180,E1 -19097.638,E2 -19097.638} C_VEL
LIN {X 0,Y 246.989,Z 653.722,A -85,B 0,C 180,E1 -19098.959,E2 -19098.959} C_VEL
LIN {X 0,Y 243.131,Z 654.196,A -85,B 0,C 180,E1 -19101.618,E2 -19101.618} C_VEL
LIN {X 0,Y 242.081,Z 654.33,A -85,B 0,C 180,E1 -19103.008,E2 -19103.008} C_VEL
LIN {X 0,Y 242.018,Z 654.333,A -85,B 0,C 180,E1 -19103.48,E2 -19103.48} C_VEL
LIN {X 0,Y 242.064,Z 654.33,A -85,B 0,C 180,E1 -19105.838,E2 -19105.838} C_VEL
LIN {X 0,Y 242.026,Z 654.339,A -85,B 0,C 180,E1 -19109.581,E2 -19109.581} C_VEL
LIN {X 0,Y 241.985,Z 654.34,A -85,B 0,C 180,E1 -19113.492,E2 -19113.492} C_VEL
LIN {X 0,Y 241.988,Z 654.339,A -85,B 0,C 180,E1 -19117.582,E2 -19117.582} C_VEL
LIN {X 0,Y 241.988,Z 654.342,A -85,B 0,C 180,E1 -19122.688,E2 -19122.688} C_VEL
LIN {X 0,Y 242.052,Z 654.592,A -85,B 0,C 180,E1 -19123.46,E2 -19123.46} C_VEL
LIN {X 0,Y 242.549,Z 657.386,A -85,B 0,C 180,E1 -19126.418,E2 -19126.418} C_VEL
LIN {X 0,Y 243.412,Z 662.145,A -85,B 0,C 180,E1 -19131.221,E2 -19131.221} C_VEL
LIN {X 0,Y 243.511,Z 664.99,A -85,B 0,C 180,E1 -19133.912,E2 -19133.912} C_VEL
LIN {X 0,Y 243.311,Z 666.176,A -85,B 0,C 180,E1 -19134.949,E2 -19134.949} C_VEL
LIN {X 0,Y 244.123,Z 669.348,A -85,B 0,C 180,E1 -19135.309,E2 -19135.309} C_VEL
LIN {X 0,Y 245.405,Z 672.213,A -85,B 0,C 180,E1 -19135.771,E2 -19135.771} C_VEL
LIN {X 0,Y 249.583,Z 684.892,A -85,B 0,C 180,E1 -19137.596,E2 -19137.596} C_VEL
LIN {X 0,Y 252.218,Z 696.457,A -85,B 0,C 180,E1 -19139.264,E2 -19139.264} C_VEL
LIN {X 0,Y 253.867,Z 708.511,A -85,B 0,C 180,E1 -19141.093,E2 -19141.093} C_VEL
LIN {X 0,Y 254.274,Z 719.281,A -85,B 0,C 180,E1 -19142.853,E2 -19142.853} C_VEL
LIN {X 0,Y 253.601,Z 729.976,A -85,B 0,C 180,E1 -19144.782,E2 -19144.782} C_VEL
LIN {X 0,Y 251.252,Z 738.995,A -85,B 0,C 180,E1 -19146.51,E2 -19146.51} C_VEL
LIN {X 0,Y 248.279,Z 748.779,A -85,B 0,C 180,E1 -19148.845,E2 -19148.845} C_VEL
LIN {X 0,Y 245.89,Z 756.733,A -85,B 0,C 180,E1 -19151.261,E2 -19151.261} C_VEL
LIN {X 0,Y 244.194,Z 762.097,A -85,B 0,C 180,E1 -19153.274,E2 -19153.274} C_VEL
LIN {X 0,Y 242.443,Z 767.442,A -85,B 0,C 180,E1 -19155.736,E2 -19155.736} C_VEL
LIN {X 0,Y 241.231,Z 771.626,A -85,B 0,C 180,E1 -19158.234,E2 -19158.234} C_VEL
LIN {X 0,Y 240.668,Z 773.851,A -85,B 0,C 180,E1 -19159.91,E2 -19159.91} C_VEL
LIN {X 0,Y 239.959,Z 776.945,A -85,B 0,C 180,E1 -19163.273,E2 -19163.273} C_VEL
LIN {X 0,Y 239.841,Z 777.956,A -85,B 0,C 180,E1 -19165.066,E2 -19165.066} C_VEL
LIN {X 0,Y 239.916,Z 779.731,A -85,B 0,C 180,E1 -19170.001,E2 -19170.001} C_VEL
LIN {X 0,Y 239.838,Z 780.015,A -85,B 0,C 180,E1 -19171.68,E2 -19171.68} C_VEL
LIN {X 0,Y 239.836,Z 779.457,A -85,B 0,C 180,E1 -19174.918,E2 -19174.918} C_VEL
LIN {X 0,Y 239.995,Z 778.468,A -85,B 0,C 180,E1 -19176.727,E2 -19176.727} C_VEL
LIN {X 0,Y 240.685,Z 775.416,A -85,B 0,C 180,E1 -19180.091,E2 -19180.091} C_VEL
LIN {X 0,Y 241.653,Z 771.987,A -85,B 0,C 180,E1 -19182.599,E2 -19182.599} C_VEL
LIN {X 0,Y 243.003,Z 767.534,A -85,B 0,C 180,E1 -19185.088,E2 -19185.088} C_VEL
LIN {X 0,Y 245.366,Z 760.868,A -85,B 0,C 180,E1 -19187.934,E2 -19187.934} C_VEL
LIN {X 0,Y 247.725,Z 752.935,A -85,B 0,C 180,E1 -19190.574,E2 -19190.574} C_VEL
LIN {X 0,Y 250.227,Z 744.81,A -85,B 0,C 180,E1 -19192.718,E2 -19192.718} C_VEL
LIN {X 0,Y 253.262,Z 734.767,A -85,B 0,C 180,E1 -19194.817,E2 -19194.817} C_VEL
LIN {X 0,Y 254.478,Z 729.472,A -85,B 0,C 180,E1 -19195.784,E2 -19195.784} C_VEL
LIN {X 0,Y 254.866,Z 720.848,A -85,B 0,C 180,E1 -19197.371,E2 -19197.371} C_VEL
LIN {X 0,Y 254.385,Z 711.012,A -85,B 0,C 180,E1 -19199.046,E2 -19199.046} C_VEL
LIN {X 0,Y 252.709,Z 699.775,A -85,B 0,C 180,E1 -19200.86,E2 -19200.86} C_VEL
LIN {X 0,Y 249.695,Z 688.001,A -85,B 0,C 180,E1 -19202.738,E2 -19202.738} C_VEL
LIN {X 0,Y 246.789,Z 679.865,A -85,B 0,C 180,E1 -19204.08,E2 -19204.08} C_VEL
LIN {X 0,Y 245.388,Z 676.287,A -85,B 0,C 180,E1 -19204.666,E2 -19204.666} C_VEL
LIN {X 0,Y 244.121,Z 673.261,A -85,B 0,C 180,E1 -19205.176,E2 -19205.176} C_VEL
LIN {X 0,Y 243.922,Z 672.139,A -85,B 0,C 180,E1 -19205.325,E2 -19205.325} C_VEL
LIN {X 0,Y 244.147,Z 670.406,A -85,B 0,C 180,E1 -19207.194,E2 -19207.194} C_VEL
LIN {X 0,Y 244.189,Z 668.607,A -85,B 0,C 180,E1 -19209.286,E2 -19209.286} C_VEL
LIN {X 0,Y 244.024,Z 666.823,A -85,B 0,C 180,E1 -19211.512,E2 -19211.512} C_VEL
LIN {X 0,Y 243.833,Z 665.05,A -85,B 0,C 180,E1 -19213.898,E2 -19213.898} C_VEL
LIN {X 0,Y 243.319,Z 662.12,A -85,B 0,C 180,E1 -19218.369,E2 -19218.369} C_VEL
LIN {X 0,Y 242.952,Z 659.791,A -85,B 0,C 180,E1 -19222.593,E2 -19222.593} C_VEL
LIN {X 0,Y 242.627,Z 658.002,A -85,B 0,C 180,E1 -19226.608,E2 -19226.608} C_VEL
LIN {X 0,Y 242.452,Z 656.658,A -85,B 0,C 180,E1 -19230.476,E2 -19230.476} C_VEL
LIN {X 0,Y 242.327,Z 655.728,A -85,B 0,C 180,E1 -19234.213,E2 -19234.213} C_VEL
LIN {X 0,Y 242.191,Z 655.146,A -85,B 0,C 180,E1 -19238.217,E2 -19238.217} C_VEL
LIN {X 0,Y 242.262,Z 654.962,A -85,B 0,C 180,E1 -19243.203,E2 -19243.203} C_VEL
LIN {X 0,Y 242.354,Z 655.191,A -85,B 0,C 180,E1 -19246.586,E2 -19246.586} C_VEL
LIN {X 0,Y 242.597,Z 655.684,A -85,B 0,C 180,E1 -19250.058,E2 -19250.058} C_VEL
LIN {X 0,Y 242.771,Z 656.428,A -85,B 0,C 180,E1 -19253.35,E2 -19253.35} C_VEL
LIN {X 0,Y 243.232,Z 657.977,A -85,B 0,C 180,E1 -19258.344,E2 -19258.344} C_VEL
LIN {X 0,Y 243.436,Z 658.589,A -85,B 0,C 180,E1 -19260,E2 -19260} C_VEL
LIN {X 0,Y 243.361,Z 660.904,A -85,B 0,C 180,E1 -19264.97,E2 -19264.97} C_VEL
LIN {X 0,Y 243.329,Z 662.705,A -85,B 0,C 180,E1 -19268.303,E2 -19268.303} C_VEL
LIN {X 0,Y 243.302,Z 663.642,A -85,B 0,C 180,E1 -19269.666,E2 -19269.666} C_VEL
LIN {X 0,Y 244.358,Z 666.625,A -85,B 0,C 180,E1 -19270.136,E2 -19270.136} C_VEL
LIN {X 0,Y 245.639,Z 668.971,A -85,B 0,C 180,E1 -19270.617,E2 -19270.617} C_VEL
LIN {X 0,Y 249.067,Z 676.741,A -85,B 0,C 180,E1 -19272.087,E2 -19272.087} C_VEL
LIN {X 0,Y 252.618,Z 686.633,A -85,B 0,C 180,E1 -19273.884,E2 -19273.884} C_VEL
LIN {X 0,Y 255.186,Z 696.618,A -85,B 0,C 180,E1 -19275.695,E2 -19275.695} C_VEL
LIN {X 0,Y 256.704,Z 706.567,A -85,B 0,C 180,E1 -19277.527,E2 -19277.527} C_VEL
LIN {X 0,Y 257.091,Z 711.753,A -85,B 0,C 180,E1 -19278.529,E2 -19278.529} C_VEL
LIN {X 0,Y 255.098,Z 720.218,A -85,B 0,C 180,E1 -19279.956,E2 -19279.956} C_VEL
LIN {X 0,Y 252.062,Z 730.751,A -85,B 0,C 180,E1 -19282.111,E2 -19282.111} C_VEL
LIN {X 0,Y 249.567,Z 738.561,A -85,B 0,C 180,E1 -19284.1,E2 -19284.1} C_VEL
LIN {X 0,Y 246.937,Z 746.438,A -85,B 0,C 180,E1 -19286.632,E2 -19286.632} C_VEL
LIN {X 0,Y 244.718,Z 752.74,A -85,B 0,C 180,E1 -19289.224,E2 -19289.224} C_VEL
LIN {X 0,Y 242.831,Z 758.015,A -85,B 0,C 180,E1 -19292.061,E2 -19292.061} C_VEL
LIN {X 0,Y 241.663,Z 761.259,A -85,B 0,C 180,E1 -19294.417,E2 -19294.417} C_VEL
LIN {X 0,Y 241.192,Z 762.6,A -85,B 0,C 180,E1 -19295.646,E2 -19295.646} C_VEL
LIN {X 0,Y 240.476,Z 764.473,A -85,B 0,C 180,E1 -19297.899,E2 -19297.899} C_VEL
LIN {X 0,Y 239.912,Z 765.697,A -85,B 0,C 180,E1 -19300.39,E2 -19300.39} C_VEL
LIN {X 0,Y 239.597,Z 766.054,A -85,B 0,C 180,E1 -19302.834,E2 -19302.834} C_VEL
LIN {X 0,Y 239.495,Z 765.561,A -85,B 0,C 180,E1 -19305.228,E2 -19305.228} C_VEL
LIN {X 0,Y 239.646,Z 764.287,A -85,B 0,C 180,E1 -19307.583,E2 -19307.583} C_VEL
LIN {X 0,Y 239.895,Z 762.29,A -85,B 0,C 180,E1 -19309.87,E2 -19309.87} C_VEL
LIN {X 0,Y 240.261,Z 759.487,A -85,B 0,C 180,E1 -19312.166,E2 -19312.166} C_VEL
LIN {X 0,Y 240.949,Z 755.228,A -85,B 0,C 180,E1 -19314.757,E2 -19314.757} C_VEL
LIN {X 0,Y 241.875,Z 749.514,A -85,B 0,C 180,E1 -19317.42,E2 -19317.42} C_VEL
LIN {X 0,Y 243.245,Z 742.208,A -85,B 0,C 180,E1 -19320.087,E2 -19320.087} C_VEL
LIN {X 0,Y 244.959,Z 733.18,A -85,B 0,C 180,E1 -19322.674,E2 -19322.674} C_VEL
LIN {X 0,Y 246.843,Z 723.321,A -85,B 0,C 180,E1 -19324.907,E2 -19324.907} C_VEL
LIN {X 0,Y 248.538,Z 713.627,A -85,B 0,C 180,E1 -19326.678,E2 -19326.678} C_VEL
LIN {X 0,Y 249.929,Z 703.987,A -85,B 0,C 180,E1 -19328.12,E2 -19328.12} C_VEL
LIN {X 0,Y 248.306,Z 692.673,A -85,B 0,C 180,E1 -19329.712,E2 -19329.712} C_VEL
LIN {X 0,Y 246.166,Z 681.409,A -85,B 0,C 180,E1 -19331.049,E2 -19331.049} C_VEL
LIN {X 0,Y 242.918,Z 667.936,A -85,B 0,C 180,E1 -19332.375,E2 -19332.375} C_VEL
LIN {X 0,Y 241.175,Z 661.193,A -85,B 0,C 180,E1 -19332.941,E2 -19332.941} C_VEL
LIN {X 0,Y 241.585,Z 658.108,A -85,B 0,C 180,E1 -19336.542,E2 -19336.542} C_VEL
LIN {X 0,Y 242.261,Z 654.307,A -85,B 0,C 180,E1 -19341.323,E2 -19341.323} C_VEL
LIN {X 0,Y 242.402,Z 654.29,A -85,B 0,C 180,E1 -19343.34,E2 -19343.34} C_VEL
LIN {X 0,Y 242.639,Z 654.258,A -85,B 0,C 180,E1 -19348.34,E2 -19348.34} C_VEL
LIN {X 0,Y 242.639,Z 654.256,A -85,B 0,C 180,E1 -19351.659,E2 -19351.659} C_VEL
LIN {X 0,Y 242.332,Z 654.3,A -85,B 0,C 180,E1 -19356.661,E2 -19356.661} C_VEL
LIN {X 0,Y 241.951,Z 654.346,A -85,B 0,C 180,E1 -19360.036,E2 -19360.036} C_VEL
LIN {X 0,Y 241.676,Z 654.445,A -85,B 0,C 180,E1 -19361.745,E2 -19361.745} C_VEL
LIN {X 0,Y 241.096,Z 659.685,A -85,B 0,C 180,E1 -19366.207,E2 -19366.207} C_VEL
LIN {X 0,Y 244.547,Z 673.361,A -85,B 0,C 180,E1 -19367.347,E2 -19367.347} C_VEL
LIN {X 0,Y 247.189,Z 685.823,A -85,B 0,C 180,E1 -19368.653,E2 -19368.653} C_VEL
LIN {X 0,Y 249.169,Z 698.018,A -85,B 0,C 180,E1 -19370.213,E2 -19370.213} C_VEL
LIN {X 0,Y 249.811,Z 704.334,A -85,B 0,C 180,E1 -19371.127,E2 -19371.127} C_VEL
LIN {X 0,Y 248.268,Z 714.236,A -85,B 0,C 180,E1 -19372.62,E2 -19372.62} C_VEL
LIN {X 0,Y 246.571,Z 723.906,A -85,B 0,C 180,E1 -19374.423,E2 -19374.423} C_VEL
LIN {X 0,Y 244.712,Z 733.742,A -85,B 0,C 180,E1 -19376.699,E2 -19376.699} C_VEL
LIN {X 0,Y 243.214,Z 741.556,A -85,B 0,C 180,E1 -19378.947,E2 -19378.947} C_VEL
LIN {X 0,Y 241.924,Z 748.677,A -85,B 0,C 180,E1 -19381.526,E2 -19381.526} C_VEL
LIN {X 0,Y 240.856,Z 754.84,A -85,B 0,C 180,E1 -19384.384,E2 -19384.384} C_VEL
LIN {X 0,Y 240.21,Z 758.749,A -85,B 0,C 180,E1 -19386.755,E2 -19386.755} C_VEL
LIN {X 0,Y 239.763,Z 761.635,A -85,B 0,C 180,E1 -19389.065,E2 -19389.065} C_VEL
LIN {X 0,Y 239.417,Z 764.406,A -85,B 0,C 180,E1 -19392.465,E2 -19392.465} C_VEL
LIN {X 0,Y 239.459,Z 765.4,A -85,B 0,C 180,E1 -19395.22,E2 -19395.22} C_VEL
LIN {X 0,Y 239.673,Z 765.416,A -85,B 0,C 180,E1 -19397.589,E2 -19397.589} C_VEL
LIN {X 0,Y 240.045,Z 764.636,A -85,B 0,C 180,E1 -19399.901,E2 -19399.901} C_VEL
LIN {X 0,Y 241.065,Z 762.104,A -85,B 0,C 180,E1 -19403.298,E2 -19403.298} C_VEL
LIN {X 0,Y 242.561,Z 757.974,A -85,B 0,C 180,E1 -19406.598,E2 -19406.598} C_VEL
LIN {X 0,Y 244.441,Z 752.508,A -85,B 0,C 180,E1 -19409.601,E2 -19409.601} C_VEL
LIN {X 0,Y 246.944,Z 745.33,A -85,B 0,C 180,E1 -19412.536,E2 -19412.536} C_VEL
LIN {X 0,Y 249.486,Z 737.456,A -85,B 0,C 180,E1 -19415.004,E2 -19415.004} C_VEL
LIN {X 0,Y 252.155,Z 728.806,A -85,B 0,C 180,E1 -19417.158,E2 -19417.158} C_VEL
LIN {X 0,Y 254.765,Z 719.676,A -85,B 0,C 180,E1 -19418.984,E2 -19418.984} C_VEL
LIN {X 0,Y 256.543,Z 712.687,A -85,B 0,C 180,E1 -19420.146,E2 -19420.146} C_VEL
LIN {X 0,Y 256.68,Z 708.955,A -85,B 0,C 180,E1 -19420.818,E2 -19420.818} C_VEL
LIN {X 0,Y 255.859,Z 700.171,A -85,B 0,C 180,E1 -19422.413,E2 -19422.413} C_VEL
LIN {X 0,Y 253.84,Z 689.605,A -85,B 0,C 180,E1 -19424.236,E2 -19424.236} C_VEL
LIN {X 0,Y 250.999,Z 679.739,A -85,B 0,C 180,E1 -19425.916,E2 -19425.916} C_VEL
LIN {X 0,Y 247.025,Z 669.469,A -85,B 0,C 180,E1 -19427.679,E2 -19427.679} C_VEL
LIN {X 0,Y 244.737,Z 664.761,A -85,B 0,C 180,E1 -19428.551,E2 -19428.551} C_VEL
LIN {X 0,Y 243.221,Z 661.388,A -85,B 0,C 180,E1 -19429.13,E2 -19429.13} C_VEL
LIN {X 0,Y 243.123,Z 660.922,A -85,B 0,C 180,E1 -19429.204,E2 -19429.204} C_VEL
LIN {X 0,Y 243.104,Z 658.565,A -85,B 0,C 180,E1 -19431.689,E2 -19431.689} C_VEL
LIN {X 0,Y 242.531,Z 655.682,A -85,B 0,C 180,E1 -19435.013,E2 -19435.013} C_VEL
LIN {X 0,Y 242.373,Z 654.296,A -85,B 0,C 180,E1 -19436.675,E2 -19436.675} C_VEL
LIN {X 0,Y 242.634,Z 654.263,A -85,B 0,C 180,E1 -19438.34,E2 -19438.34} C_VEL
LIN {X 0,Y 242.634,Z 654.262,A -85,B 0,C 180,E1 -19441.66,E2 -19441.66} C_VEL
LIN {X 0,Y 242.431,Z 654.289,A -85,B 0,C 180,E1 -19446.659,E2 -19446.659} C_VEL
LIN {X 0,Y 242.342,Z 654.296,A -85,B 0,C 180,E1 -19450.021,E2 -19450.021} C_VEL
LIN {X 0,Y 242.163,Z 654.321,A -85,B 0,C 180,E1 -19455.141,E2 -19455.141} C_VEL
LIN {X 0,Y 242.07,Z 654.33,A -85,B 0,C 180,E1 -19458.624,E2 -19458.624} C_VEL
LIN {X 0,Y 242.01,Z 654.339,A -85,B 0,C 180,E1 -19462.18,E2 -19462.18} C_VEL
LIN {X 0,Y 242.018,Z 654.333,A -85,B 0,C 180,E1 -19463.48,E2 -19463.48} C_VEL
LIN {X 0,Y 241.407,Z 654.415,A -85,B 0,C 180,E1 -19464.868,E2 -19464.868} C_VEL
LIN {X 0,Y 238.563,Z 654.773,A -85,B 0,C 180,E1 -19467.131,E2 -19467.131} C_VEL
LIN {X 0,Y 236.094,Z 655.079,A -85,B 0,C 180,E1 -19468.976,E2 -19468.976} C_VEL
LIN {X 0,Y 235.012,Z 655.21,A -85,B 0,C 180,E1 -19470.408,E2 -19470.408} C_VEL
LIN {X 0,Y 234.913,Z 655.219,A -85,B 0,C 180,E1 -19470.894,E2 -19470.894} C_VEL
LIN {X 0,Y 234.939,Z 655.221,A -85,B 0,C 180,E1 -19474.637,E2 -19474.637} C_VEL
LIN {X 0,Y 234.939,Z 655.221,A -85,B 0,C 180,E1 -19478.945,E2 -19478.945} C_VEL
LIN {X 0,Y 234.96,Z 655.243,A -85,B 0,C 180,E1 -19482.952,E2 -19482.952} C_VEL
LIN {X 0,Y 235.576,Z 658.652,A -85,B 0,C 180,E1 -19486.674,E2 -19486.674} C_VEL
LIN {X 0,Y 236.37,Z 663.202,A -85,B 0,C 180,E1 -19491.363,E2 -19491.363} C_VEL
LIN {X 0,Y 236.458,Z 665.209,A -85,B 0,C 180,E1 -19493.195,E2 -19493.195} C_VEL
LIN {X 0,Y 237.449,Z 668.499,A -85,B 0,C 180,E1 -19493.648,E2 -19493.648} C_VEL
LIN {X 0,Y 238.802,Z 671.302,A -85,B 0,C 180,E1 -19494.17,E2 -19494.17} C_VEL
LIN {X 0,Y 241.096,Z 677.863,A -85,B 0,C 180,E1 -19495.186,E2 -19495.186} C_VEL
LIN {X 0,Y 243.978,Z 687.146,A -85,B 0,C 180,E1 -19496.654,E2 -19496.654} C_VEL
LIN {X 0,Y 246.46,Z 698.924,A -85,B 0,C 180,E1 -19498.489,E2 -19498.489} C_VEL
LIN {X 0,Y 247.758,Z 709.773,A -85,B 0,C 180,E1 -19500.248,E2 -19500.248} C_VEL
LIN {X 0,Y 248.044,Z 720.559,A -85,B 0,C 180,E1 -19502.113,E2 -19502.113} C_VEL
LIN {X 0,Y 247.236,Z 730.95,A -85,B 0,C 180,E1 -19504.085,E2 -19504.085} C_VEL
LIN {X 0,Y 244.218,Z 741.436,A -85,B 0,C 180,E1 -19506.242,E2 -19506.242} C_VEL
LIN {X 0,Y 241.661,Z 749.431,A -85,B 0,C 180,E1 -19508.281,E2 -19508.281} C_VEL
LIN {X 0,Y 239.155,Z 757.2,A -85,B 0,C 180,E1 -19510.745,E2 -19510.745} C_VEL
LIN {X 0,Y 236.777,Z 764.246,A -85,B 0,C 180,E1 -19513.623,E2 -19513.623} C_VEL
LIN {X 0,Y 235.038,Z 769.079,A -85,B 0,C 180,E1 -19516.161,E2 -19516.161} C_VEL
LIN {X 0,Y 233.928,Z 772.812,A -85,B 0,C 180,E1 -19518.74,E2 -19518.74} C_VEL
LIN {X 0,Y 233.198,Z 775.557,A -85,B 0,C 180,E1 -19521.334,E2 -19521.334} C_VEL
LIN {X 0,Y 232.766,Z 777.783,A -85,B 0,C 180,E1 -19524.804,E2 -19524.804} C_VEL
LIN {X 0,Y 232.774,Z 778.73,A -85,B 0,C 180,E1 -19528.271,E2 -19528.271} C_VEL
LIN {X 0,Y 232.847,Z 779.464,A -85,B 0,C 180,E1 -19530.001,E2 -19530.001} C_VEL
LIN {X 0,Y 232.75,Z 779.783,A -85,B 0,C 180,E1 -19531.731,E2 -19531.731} C_VEL
LIN {X 0,Y 232.768,Z 779.255,A -85,B 0,C 180,E1 -19535.198,E2 -19535.198} C_VEL
LIN {X 0,Y 232.922,Z 778.374,A -85,B 0,C 180,E1 -19536.933,E2 -19536.933} C_VEL
LIN {X 0,Y 233.683,Z 775.406,A -85,B 0,C 180,E1 -19540.397,E2 -19540.397} C_VEL
LIN {X 0,Y 234.714,Z 772.074,A -85,B 0,C 180,E1 -19542.978,E2 -19542.978} C_VEL
LIN {X 0,Y 236.162,Z 767.709,A -85,B 0,C 180,E1 -19545.536,E2 -19545.536} C_VEL
LIN {X 0,Y 238.627,Z 761.177,A -85,B 0,C 180,E1 -19548.458,E2 -19548.458} C_VEL
LIN {X 0,Y 241.005,Z 753.695,A -85,B 0,C 180,E1 -19551.067,E2 -19551.067} C_VEL
LIN {X 0,Y 243.738,Z 745.423,A -85,B 0,C 180,E1 -19553.358,E2 -19553.358} C_VEL
LIN {X 0,Y 246.585,Z 736.616,A -85,B 0,C 180,E1 -19555.311,E2 -19555.311} C_VEL
LIN {X 0,Y 248.135,Z 730.506,A -85,B 0,C 180,E1 -19556.494,E2 -19556.494} C_VEL
LIN {X 0,Y 248.628,Z 722.096,A -85,B 0,C 180,E1 -19558.118,E2 -19558.118} C_VEL
LIN {X 0,Y 248.259,Z 712.392,A -85,B 0,C 180,E1 -19559.875,E2 -19559.875} C_VEL
LIN {X 0,Y 246.861,Z 701.964,A -85,B 0,C 180,E1 -19561.683,E2 -19561.683} C_VEL
LIN {X 0,Y 243.914,Z 689.836,A -85,B 0,C 180,E1 -19563.762,E2 -19563.762} C_VEL
LIN {X 0,Y 240.704,Z 680.685,A -85,B 0,C 180,E1 -19565.403,E2 -19565.403} C_VEL
LIN {X 0,Y 238.829,Z 676.202,A -85,B 0,C 180,E1 -19566.231,E2 -19566.231} C_VEL
LIN {X 0,Y 237.382,Z 673.02,A -85,B 0,C 180,E1 -19566.854,E2 -19566.854} C_VEL
LIN {X 0,Y 237.146,Z 671.809,A -85,B 0,C 180,E1 -19567.039,E2 -19567.039} C_VEL
LIN {X 0,Y 237.08,Z 668.823,A -85,B 0,C 180,E1 -19570.706,E2 -19570.706} C_VEL
LIN {X 0,Y 236.783,Z 666.035,A -85,B 0,C 180,E1 -19574.574,E2 -19574.574} C_VEL
LIN {X 0,Y 236.305,Z 663.22,A -85,B 0,C 180,E1 -19579.133,E2 -19579.133} C_VEL
LIN {X 0,Y 235.959,Z 660.949,A -85,B 0,C 180,E1 -19583.533,E2 -19583.533} C_VEL
LIN {X 0,Y 235.647,Z 659.319,A -85,B 0,C 180,E1 -19587.531,E2 -19587.531} C_VEL
LIN {X 0,Y 235.473,Z 658.078,A -85,B 0,C 180,E1 -19591.475,E2 -19591.475} C_VEL
LIN {X 0,Y 235.373,Z 657.245,A -85,B 0,C 180,E1 -19595.29,E2 -19595.29} C_VEL
LIN {X 0,Y 235.269,Z 656.798,A -85,B 0,C 180,E1 -19598.994,E2 -19598.994} C_VEL
LIN {X 0,Y 235.355,Z 656.656,A -85,B 0,C 180,E1 -19602.856,E2 -19602.856} C_VEL
LIN {X 0,Y 235.45,Z 656.825,A -85,B 0,C 180,E1 -19606.185,E2 -19606.185} C_VEL
LIN {X 0,Y 235.647,Z 657.287,A -85,B 0,C 180,E1 -19609.804,E2 -19609.804} C_VEL
LIN {X 0,Y 235.844,Z 657.982,A -85,B 0,C 180,E1 -19613.154,E2 -19613.154} C_VEL
LIN {X 0,Y 236.303,Z 659.485,A -85,B 0,C 180,E1 -19618.296,E2 -19618.296} C_VEL
LIN {X 0,Y 236.496,Z 660.1,A -85,B 0,C 180,E1 -19620,E2 -19620} C_VEL
LIN {X 0,Y 236.412,Z 661.58,A -85,B 0,C 180,E1 -19623.409,E2 -19623.409} C_VEL
LIN {X 0,Y 236.372,Z 663.806,A -85,B 0,C 180,E1 -19627.85,E2 -19627.85} C_VEL
LIN {X 0,Y 237.553,Z 666.967,A -85,B 0,C 180,E1 -19628.453,E2 -19628.453} C_VEL
LIN {X 0,Y 238.944,Z 668.948,A -85,B 0,C 180,E1 -19628.99,E2 -19628.99} C_VEL
LIN {X 0,Y 243.888,Z 680.365,A -85,B 0,C 180,E1 -19631.312,E2 -19631.312} C_VEL
LIN {X 0,Y 247.013,Z 689.736,A -85,B 0,C 180,E1 -19633.157,E2 -19633.157} C_VEL
LIN {X 0,Y 249.408,Z 699.782,A -85,B 0,C 180,E1 -19635.109,E2 -19635.109} C_VEL
LIN {X 0,Y 250.676,Z 709.954,A -85,B 0,C 180,E1 -19637.121,E2 -19637.121} C_VEL
LIN {X 0,Y 250.844,Z 714.011,A -85,B 0,C 180,E1 -19637.95,E2 -19637.95} C_VEL
LIN {X 0,Y 247.88,Z 724.718,A -85,B 0,C 180,E1 -19639.891,E2 -19639.891} C_VEL
LIN {X 0,Y 245.051,Z 733.558,A -85,B 0,C 180,E1 -19641.891,E2 -19641.891} C_VEL
LIN {X 0,Y 242.128,Z 742.008,A -85,B 0,C 180,E1 -19644.283,E2 -19644.283} C_VEL
LIN {X 0,Y 239.457,Z 749.388,A -85,B 0,C 180,E1 -19646.963,E2 -19646.963} C_VEL
LIN {X 0,Y 237.568,Z 754.329,A -85,B 0,C 180,E1 -19649.217,E2 -19649.217} C_VEL
LIN {X 0,Y 236.081,Z 758.212,A -85,B 0,C 180,E1 -19651.447,E2 -19651.447} C_VEL
LIN {X 0,Y 234.46,Z 762.391,A -85,B 0,C 180,E1 -19654.718,E2 -19654.718} C_VEL
LIN {X 0,Y 233.618,Z 764.39,A -85,B 0,C 180,E1 -19656.99,E2 -19656.99} C_VEL
LIN {X 0,Y 233.006,Z 765.65,A -85,B 0,C 180,E1 -19659.302,E2 -19659.302} C_VEL
LIN {X 0,Y 232.627,Z 766.224,A -85,B 0,C 180,E1 -19661.656,E2 -19661.656} C_VEL
LIN {X 0,Y 232.409,Z 766.078,A -85,B 0,C 180,E1 -19664.069,E2 -19664.069} C_VEL
LIN {X 0,Y 232.44,Z 765.108,A -85,B 0,C 180,E1 -19666.524,E2 -19666.524} C_VEL
LIN {X 0,Y 232.689,Z 763.266,A -85,B 0,C 180,E1 -19669.033,E2 -19669.033} C_VEL
LIN {X 0,Y 233.066,Z 760.424,A -85,B 0,C 180,E1 -19671.63,E2 -19671.63} C_VEL
LIN {X 0,Y 233.701,Z 756.436,A -85,B 0,C 180,E1 -19674.288,E2 -19674.288} C_VEL
LIN {X 0,Y 234.756,Z 750.221,A -85,B 0,C 180,E1 -19677.392,E2 -19677.392} C_VEL
LIN {X 0,Y 236.175,Z 742.735,A -85,B 0,C 180,E1 -19680.237,E2 -19680.237} C_VEL
LIN {X 0,Y 237.659,Z 735.218,A -85,B 0,C 180,E1 -19682.518,E2 -19682.518} C_VEL
LIN {X 0,Y 239.312,Z 726.901,A -85,B 0,C 180,E1 -19684.579,E2 -19684.579} C_VEL
LIN {X 0,Y 241.197,Z 716.75,A -85,B 0,C 180,E1 -19686.608,E2 -19686.608} C_VEL
LIN {X 0,Y 243.022,Z 705.782,A -85,B 0,C 180,E1 -19688.363,E2 -19688.363} C_VEL
LIN {X 0,Y 241.888,Z 696.094,A -85,B 0,C 180,E1 -19689.816,E2 -19689.816} C_VEL
LIN {X 0,Y 239.651,Z 683.747,A -85,B 0,C 180,E1 -19691.408,E2 -19691.408} C_VEL
LIN {X 0,Y 236.444,Z 670.12,A -85,B 0,C 180,E1 -19692.841,E2 -19692.841} C_VEL
LIN {X 0,Y 234.227,Z 661.382,A -85,B 0,C 180,E1 -19693.617,E2 -19693.617} C_VEL
LIN {X 0,Y 234.679,Z 657.843,A -85,B 0,C 180,E1 -19697.899,E2 -19697.899} C_VEL
LIN {X 0,Y 235.225,Z 655.183,A -85,B 0,C 180,E1 -19701.408,E2 -19701.408} C_VEL
LIN {X 0,Y 235.345,Z 655.169,A -85,B 0,C 180,E1 -19703.139,E2 -19703.139} C_VEL
LIN {X 0,Y 235.599,Z 655.135,A -85,B 0,C 180,E1 -19708.29,E2 -19708.29} C_VEL
LIN {X 0,Y 235.598,Z 655.133,A -85,B 0,C 180,E1 -19711.709,E2 -19711.709} C_VEL
LIN {X 0,Y 235.27,Z 655.177,A -85,B 0,C 180,E1 -19716.862,E2 -19716.862} C_VEL
LIN {X 0,Y 234.864,Z 655.229,A -85,B 0,C 180,E1 -19720.342,E2 -19720.342} C_VEL
LIN {X 0,Y 234.649,Z 655.338,A -85,B 0,C 180,E1 -19721.663,E2 -19721.663} C_VEL
LIN {X 0,Y 234.107,Z 659.676,A -85,B 0,C 180,E1 -19725.507,E2 -19725.507} C_VEL
LIN {X 0,Y 237.767,Z 674.249,A -85,B 0,C 180,E1 -19726.788,E2 -19726.788} C_VEL
LIN {X 0,Y 240.275,Z 686.242,A -85,B 0,C 180,E1 -19728.105,E2 -19728.105} C_VEL
LIN {X 0,Y 242.303,Z 698.828,A -85,B 0,C 180,E1 -19729.781,E2 -19729.781} C_VEL
LIN {X 0,Y 242.94,Z 705.199,A -85,B 0,C 180,E1 -19730.742,E2 -19730.742} C_VEL
LIN {X 0,Y 241.094,Z 716.183,A -85,B 0,C 180,E1 -19732.494,E2 -19732.494} C_VEL
LIN {X 0,Y 239.304,Z 725.959,A -85,B 0,C 180,E1 -19734.435,E2 -19734.435} C_VEL
LIN {X 0,Y 237.463,Z 735.443,A -85,B 0,C 180,E1 -19736.78,E2 -19736.78} C_VEL
LIN {X 0,Y 235.892,Z 743.349,A -85,B 0,C 180,E1 -19739.235,E2 -19739.235} C_VEL
LIN {X 0,Y 234.554,Z 750.721,A -85,B 0,C 180,E1 -19742.129,E2 -19742.129} C_VEL
LIN {X 0,Y 233.615,Z 756.055,A -85,B 0,C 180,E1 -19744.86,E2 -19744.86} C_VEL
LIN {X 0,Y 233.03,Z 759.483,A -85,B 0,C 180,E1 -19747.097,E2 -19747.097} C_VEL
LIN {X 0,Y 232.611,Z 762.13,A -85,B 0,C 180,E1 -19749.381,E2 -19749.381} C_VEL
LIN {X 0,Y 232.33,Z 764.061,A -85,B 0,C 180,E1 -19751.72,E2 -19751.72} C_VEL
LIN {X 0,Y 232.33,Z 765.26,A -85,B 0,C 180,E1 -19754.086,E2 -19754.086} C_VEL
LIN {X 0,Y 232.44,Z 765.72,A -85,B 0,C 180,E1 -19756.522,E2 -19756.522} C_VEL
LIN {X 0,Y 232.791,Z 765.348,A -85,B 0,C 180,E1 -19759.002,E2 -19759.002} C_VEL
LIN {X 0,Y 233.359,Z 764.125,A -85,B 0,C 180,E1 -19761.538,E2 -19761.538} C_VEL
LIN {X 0,Y 234.286,Z 762.007,A -85,B 0,C 180,E1 -19764.088,E2 -19764.088} C_VEL
LIN {X 0,Y 235.491,Z 758.882,A -85,B 0,C 180,E1 -19766.68,E2 -19766.68} C_VEL
LIN {X 0,Y 237.432,Z 753.694,A -85,B 0,C 180,E1 -19769.788,E2 -19769.788} C_VEL
LIN {X 0,Y 239.673,Z 747.578,A -85,B 0,C 180,E1 -19772.494,E2 -19772.494} C_VEL
LIN {X 0,Y 242.597,Z 739.438,A -85,B 0,C 180,E1 -19775.285,E2 -19775.285} C_VEL
LIN {X 0,Y 245.396,Z 730.935,A -85,B 0,C 180,E1 -19777.557,E2 -19777.557} C_VEL
LIN {X 0,Y 248.629,Z 720.382,A -85,B 0,C 180,E1 -19779.775,E2 -19779.775} C_VEL
LIN {X 0,Y 250.522,Z 712.348,A -85,B 0,C 180,E1 -19781.179,E2 -19781.179} C_VEL
LIN {X 0,Y 249.875,Z 702.997,A -85,B 0,C 180,E1 -19782.993,E2 -19782.993} C_VEL
LIN {X 0,Y 248.264,Z 693.182,A -85,B 0,C 180,E1 -19784.82,E2 -19784.82} C_VEL
LIN {X 0,Y 245.392,Z 682.606,A -85,B 0,C 180,E1 -19786.755,E2 -19786.755} C_VEL
LIN {X 0,Y 241.807,Z 672.917,A -85,B 0,C 180,E1 -19788.573,E2 -19788.573} C_VEL
LIN {X 0,Y 239.98,Z 668.948,A -85,B 0,C 180,E1 -19789.353,E2 -19789.353} C_VEL
LIN {X 0,Y 238.23,Z 665.293,A -85,B 0,C 180,E1 -19790.073,E2 -19790.073} C_VEL
LIN {X 0,Y 236.415,Z 661.801,A -85,B 0,C 180,E1 -19790.806,E2 -19790.806} C_VEL
LIN {X 0,Y 236.243,Z 661.145,A -85,B 0,C 180,E1 -19790.907,E2 -19790.907} C_VEL
LIN {X 0,Y 236.078,Z 659.17,A -85,B 0,C 180,E1 -19793.161,E2 -19793.161} C_VEL
LIN {X 0,Y 235.594,Z 655.14,A -85,B 0,C 180,E1 -19798.29,E2 -19798.29} C_VEL
LIN {X 0,Y 235.594,Z 655.139,A -85,B 0,C 180,E1 -19801.709,E2 -19801.709} C_VEL
LIN {X 0,Y 235.403,Z 655.163,A -85,B 0,C 180,E1 -19806.859,E2 -19806.859} C_VEL
LIN {X 0,Y 235.25,Z 655.181,A -85,B 0,C 180,E1 -19810.326,E2 -19810.326} C_VEL
LIN {X 0,Y 235.111,Z 655.2,A -85,B 0,C 180,E1 -19815.607,E2 -19815.607} C_VEL
LIN {X 0,Y 235.006,Z 655.209,A -85,B 0,C 180,E1 -19819.206,E2 -19819.206} C_VEL
LIN {X 0,Y 234.939,Z 655.217,A -85,B 0,C 180,E1 -19823.476,E2 -19823.476} C_VEL
LIN {X 0,Y 234.967,Z 655.214,A -85,B 0,C 180,E1 -19826.658,E2 -19826.658} C_VEL
LIN {X 0,Y 234.913,Z 655.219,A -85,B 0,C 180,E1 -19830.894,E2 -19830.894} C_VEL
LIN {X 0,Y 234.219,Z 655.311,A -85,B 0,C 180,E1 -19832.326,E2 -19832.326} C_VEL
LIN {X 0,Y 231.363,Z 655.666,A -85,B 0,C 180,E1 -19834.663,E2 -19834.663} C_VEL
LIN {X 0,Y 228.951,Z 655.967,A -85,B 0,C 180,E1 -19836.568,E2 -19836.568} C_VEL
LIN {X 0,Y 227.915,Z 656.092,A -85,B 0,C 180,E1 -19838.046,E2 -19838.046} C_VEL
LIN {X 0,Y 227.829,Z 656.101,A -85,B 0,C 180,E1 -19838.548,E2 -19838.548} C_VEL
LIN {X 0,Y 227.931,Z 656.13,A -85,B 0,C 180,E1 -19842.715,E2 -19842.715} C_VEL
LIN {X 0,Y 228.68,Z 660.452,A -85,B 0,C 180,E1 -19847.527,E2 -19847.527} C_VEL
LIN {X 0,Y 229.105,Z 662.919,A -85,B 0,C 180,E1 -19849.896,E2 -19849.896} C_VEL
LIN {X 0,Y 229.533,Z 665.011,A -85,B 0,C 180,E1 -19851.248,E2 -19851.248} C_VEL
LIN {X 0,Y 230.878,Z 668.254,A -85,B 0,C 180,E1 -19851.858,E2 -19851.858} C_VEL
LIN {X 0,Y 232.27,Z 670.54,A -85,B 0,C 180,E1 -19852.406,E2 -19852.406} C_VEL
LIN {X 0,Y 234.754,Z 677.139,A -85,B 0,C 180,E1 -19853.569,E2 -19853.569} C_VEL
LIN {X 0,Y 237.154,Z 684.623,A -85,B 0,C 180,E1 -19854.864,E2 -19854.864} C_VEL
LIN {X 0,Y 239.745,Z 695.359,A -85,B 0,C 180,E1 -19856.663,E2 -19856.663} C_VEL
LIN {X 0,Y 241.413,Z 707.032,A -85,B 0,C 180,E1 -19858.642,E2 -19858.642} C_VEL
LIN {X 0,Y 241.925,Z 718.153,A -85,B 0,C 180,E1 -19860.635,E2 -19860.635} C_VEL
LIN {X 0,Y 241.407,Z 727.647,A -85,B 0,C 180,E1 -19862.474,E2 -19862.474} C_VEL
LIN {X 0,Y 240.428,Z 733.915,A -85,B 0,C 180,E1 -19863.762,E2 -19863.762} C_VEL
LIN {X 0,Y 237.249,Z 743.819,A -85,B 0,C 180,E1 -19865.965,E2 -19865.965} C_VEL
LIN {X 0,Y 234.112,Z 752.691,A -85,B 0,C 180,E1 -19868.471,E2 -19868.471} C_VEL
LIN {X 0,Y 231.742,Z 759.646,A -85,B 0,C 180,E1 -19870.974,E2 -19870.974} C_VEL
LIN {X 0,Y 229.301,Z 766.19,A -85,B 0,C 180,E1 -19873.988,E2 -19873.988} C_VEL
LIN {X 0,Y 227.698,Z 770.551,A -85,B 0,C 180,E1 -19876.616,E2 -19876.616} C_VEL
LIN {X 0,Y 226.648,Z 773.862,A -85,B 0,C 180,E1 -19879.278,E2 -19879.278} C_VEL
LIN {X 0,Y 225.827,Z 776.796,A -85,B 0,C 180,E1 -19882.85,E2 -19882.85} C_VEL
LIN {X 0,Y 225.669,Z 777.826,A -85,B 0,C 180,E1 -19885.257,E2 -19885.257} C_VEL
LIN {X 0,Y 225.687,Z 778.395,A -85,B 0,C 180,E1 -19888.216,E2 -19888.216} C_VEL
LIN {X 0,Y 225.757,Z 779.196,A -85,B 0,C 180,E1 -19890.001,E2 -19890.001} C_VEL
LIN {X 0,Y 225.664,Z 779.549,A -85,B 0,C 180,E1 -19891.785,E2 -19891.785} C_VEL
LIN {X 0,Y 225.69,Z 779.096,A -85,B 0,C 180,E1 -19895.361,E2 -19895.361} C_VEL
LIN {X 0,Y 225.847,Z 778.289,A -85,B 0,C 180,E1 -19897.151,E2 -19897.151} C_VEL
LIN {X 0,Y 226.667,Z 775.41,A -85,B 0,C 180,E1 -19900.722,E2 -19900.722} C_VEL
LIN {X 0,Y 227.762,Z 772.161,A -85,B 0,C 180,E1 -19903.382,E2 -19903.382} C_VEL
LIN {X 0,Y 229.34,Z 767.883,A -85,B 0,C 180,E1 -19906.01,E2 -19906.01} C_VEL
LIN {X 0,Y 231.911,Z 761.487,A -85,B 0,C 180,E1 -19909.013,E2 -19909.013} C_VEL
LIN {X 0,Y 234.33,Z 754.478,A -85,B 0,C 180,E1 -19911.604,E2 -19911.604} C_VEL
LIN {X 0,Y 237.284,Z 746.083,A -85,B 0,C 180,E1 -19914.033,E2 -19914.033} C_VEL
LIN {X 0,Y 240.229,Z 737.445,A -85,B 0,C 180,E1 -19916.03,E2 -19916.03} C_VEL
LIN {X 0,Y 241.837,Z 731.472,A -85,B 0,C 180,E1 -19917.24,E2 -19917.24} C_VEL
LIN {X 0,Y 242.454,Z 721.826,A -85,B 0,C 180,E1 -19919.212,E2 -19919.212} C_VEL
LIN {X 0,Y 242.016,Z 711.569,A -85,B 0,C 180,E1 -19921.168,E2 -19921.168} C_VEL
LIN {X 0,Y 240.461,Z 701.096,A -85,B 0,C 180,E1 -19923.104,E2 -19923.104} C_VEL
LIN {X 0,Y 237.839,Z 690.586,A -85,B 0,C 180,E1 -19925.066,E2 -19925.066} C_VEL
LIN {X 0,Y 234.362,Z 680.78,A -85,B 0,C 180,E1 -19926.995,E2 -19926.995} C_VEL
LIN {X 0,Y 232.393,Z 676.404,A -85,B 0,C 180,E1 -19927.939,E2 -19927.939} C_VEL
LIN {X 0,Y 230.685,Z 673.305,A -85,B 0,C 180,E1 -19928.698,E2 -19928.698} C_VEL
LIN {X 0,Y 230.191,Z 671.491,A -85,B 0,C 180,E1 -19929.004,E2 -19929.004} C_VEL
LIN {X 0,Y 230.005,Z 668.664,A -85,B 0,C 180,E1 -19932.833,E2 -19932.833} C_VEL
LIN {X 0,Y 229.567,Z 665.807,A -85,B 0,C 180,E1 -19937.286,E2 -19937.286} C_VEL
LIN {X 0,Y 229.111,Z 663.219,A -85,B 0,C 180,E1 -19942.157,E2 -19942.157} C_VEL
LIN {X 0,Y 228.866,Z 661.364,A -85,B 0,C 180,E1 -19946.445,E2 -19946.445} C_VEL
LIN {X 0,Y 228.603,Z 660.031,A -85,B 0,C 180,E1 -19950.535,E2 -19950.535} C_VEL
LIN {X 0,Y 228.499,Z 659.1,A -85,B 0,C 180,E1 -19954.494,E2 -19954.494} C_VEL
LIN {X 0,Y 228.412,Z 658.567,A -85,B 0,C 180,E1 -19958.332,E2 -19958.332} C_VEL
LIN {X 0,Y 228.472,Z 658.358,A -85,B 0,C 180,E1 -19962.477,E2 -19962.477} C_VEL
LIN {X 0,Y 228.527,Z 658.483,A -85,B 0,C 180,E1 -19965.757,E2 -19965.757} C_VEL
LIN {X 0,Y 228.704,Z 658.908,A -85,B 0,C 180,E1 -19969.532,E2 -19969.532} C_VEL
LIN {X 0,Y 228.911,Z 659.555,A -85,B 0,C 180,E1 -19972.946,E2 -19972.946} C_VEL
LIN {X 0,Y 229.38,Z 661.01,A -85,B 0,C 180,E1 -19978.244,E2 -19978.244} C_VEL
LIN {X 0,Y 229.569,Z 661.604,A -85,B 0,C 180,E1 -19980,E2 -19980} C_VEL
LIN {X 0,Y 229.466,Z 663.071,A -85,B 0,C 180,E1 -19983.512,E2 -19983.512} C_VEL
LIN {X 0,Y 229.433,Z 664.185,A -85,B 0,C 180,E1 -19985.879,E2 -19985.879} C_VEL
LIN {X 0,Y 230.607,Z 667.18,A -85,B 0,C 180,E1 -19986.508,E2 -19986.508} C_VEL
LIN {X 0,Y 232.436,Z 669.767,A -85,B 0,C 180,E1 -19987.274,E2 -19987.274} C_VEL
LIN {X 0,Y 234.3,Z 673.402,A -85,B 0,C 180,E1 -19988.163,E2 -19988.163} C_VEL
LIN {X 0,Y 238.796,Z 684.32,A -85,B 0,C 180,E1 -19990.598,E2 -19990.598} C_VEL
LIN {X 0,Y 241.38,Z 692.541,A -85,B 0,C 180,E1 -19992.341,E2 -19992.341} C_VEL
LIN {X 0,Y 243.676,Z 703.468,A -85,B 0,C 180,E1 -19994.618,E2 -19994.618} C_VEL
LIN {X 0,Y 244.6,Z 713.254,A -85,B 0,C 180,E1 -19996.698,E2 -19996.698} C_VEL
LIN {X 0,Y 244.412,Z 716.6,A -85,B 0,C 180,E1 -19997.39,E2 -19997.39} C_VEL
LIN {X 0,Y 241.371,Z 726.687,A -85,B 0,C 180,E1 -19999.342,E2 -19999.342} C_VEL
LIN {X 0,Y 238.761,Z 734.285,A -85,B 0,C 180,E1 -20001.136,E2 -20001.136} C_VEL
LIN {X 0,Y 236.061,Z 741.636,A -85,B 0,C 180,E1 -20003.257,E2 -20003.257} C_VEL
LIN {X 0,Y 233.637,Z 747.97,A -85,B 0,C 180,E1 -20005.52,E2 -20005.52} C_VEL
LIN {X 0,Y 231.215,Z 753.904,A -85,B 0,C 180,E1 -20008.177,E2 -20008.177} C_VEL
LIN {X 0,Y 228.945,Z 759.358,A -85,B 0,C 180,E1 -20011.457,E2 -20011.457} C_VEL
